KUKA KRL program: MyProgram_110().src

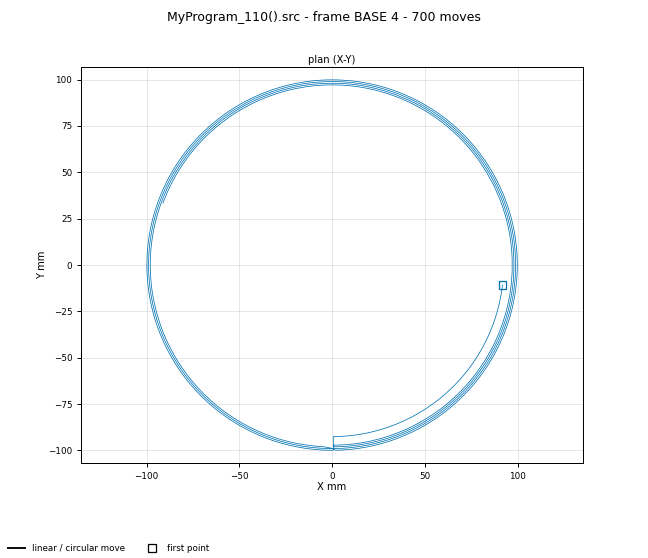
[picture p0: tool path of MyProgram_110().src in frame BASE 4, 700 of 700 moves have a stored position in this frame; points joined in program order, loops and branches not executed]
&ACCESS RVP
&REL 1
&PARAM TEMPLATE = C:\KRC\Roboter\Template\vorgabe
&PARAM EDITMASK = *
DEF MyProgram_110()
; ---- Setting reference (Base) ----
$BASE = BASE_DATA[4]

; --------------------------
; ---- Setting tool (TCP) ----
$TOOL = TOOL_DATA[3]
; --------------------------

$VEL.CP = VEL_APROX_PRINT
Startdeposition()
$VEL.CP = VEL_PRINT
LIN {X 91.8792,Y -10.8484,Z 96,A -11.884,B 24.923,C -2.0263,E1 25.1586,E2 97.0234} C_DIS
LIN {X 91.5181,Y -13.5726,Z 96,A -13.5745,B 24.9234,C -2.0212,E1 25.1579,E2 98.7159} C_DIS
LIN {X 91.0731,Y -16.2835,Z 96,A -15.3127,B 24.9239,C -2.0144,E1 25.1571,E2 100.46} C_DIS
LIN {X 90.5157,Y -19.1486,Z 96,A -17.2609,B 24.9247,C -2.0034,E1 25.156,E2 102.4228} C_DIS
LIN {X 89.7406,Y -22.5028,Z 96,A -19.3635,B 24.9252,C -1.9977,E1 25.1546,E2 104.5265} C_DIS
LIN {X 88.9858,Y -25.3177,Z 96,A -21.051,B 24.9252,C -1.9964,E1 25.1534,E2 106.2075} C_DIS
LIN {X 88.0495,Y -28.4034,Z 96,A -23.0482,B 24.9257,C -1.9901,E1 25.1517,E2 108.2082} C_DIS
LIN {X 87.1124,Y -31.1642,Z 96,A -24.7456,B 24.9259,C -1.9885,E1 25.1502,E2 109.8999} C_DIS
LIN {X 86.1483,Y -33.7335,Z 96,A -26.4825,B 24.9264,C -1.9819,E1 25.1484,E2 111.6427} C_DIS
LIN {X 85.0444,Y -36.4307,Z 96,A -28.2267,B 24.9266,C -1.9786,E1 25.1466,E2 113.3851} C_DIS
LIN {X 83.8742,Y -39.0457,Z 96,A -30.1195,B 24.9273,C -1.9689,E1 25.1444,E2 115.2905} C_DIS
LIN {X 82.3306,Y -42.2037,Z 96,A -32.231,B 24.9276,C -1.9648,E1 25.1417,E2 117.4003} C_DIS
LIN {X 80.8218,Y -45.0257,Z 96,A -34.1754,B 24.9279,C -1.9604,E1 25.1391,E2 119.345} C_DIS
LIN {X 79.3526,Y -47.5703,Z 96,A -35.9275,B 24.9282,C -1.9576,E1 25.1367,E2 121.0947} C_DIS
LIN {X 78.165,Y -49.4976,Z 96,A -37.5141,B 24.9289,C -1.9468,E1 25.1343,E2 122.6986} C_DIS
LIN {X 76.385,Y -52.2011,Z 96,A -39.5403,B 24.9294,C -1.9404,E1 25.1311,E2 124.7299} C_DIS
LIN {X 74.2916,Y -55.1408,Z 96,A -41.7416,B 24.9298,C -1.9355,E1 25.1275,E2 126.9321} C_DIS
LIN {X 72.2294,Y -57.816,Z 96,A -43.8281,B 24.9302,C -1.9302,E1 25.1239,E2 129.0215} C_DIS
LIN {X 70.1015,Y -60.3779,Z 96,A -45.7008,B 24.93,C -1.9317,E1 25.1205,E2 130.8819} C_DIS
LIN {X 68.086,Y -62.64,Z 96,A -47.6453,B 24.9306,C -1.9245,E1 25.1169,E2 132.8349} C_DIS
LIN {X 65.7943,Y -65.0428,Z 96,A -49.6815,B 24.9309,C -1.9202,E1 25.1129,E2 134.8726} C_DIS
LIN {X 63.3926,Y -67.3857,Z 96,A -51.8033,B 24.9314,C -1.9136,E1 25.1086,E2 137.0011} C_DIS
LIN {X 60.815,Y -69.7209,Z 96,A -53.9021,B 24.9316,C -1.9106,E1 25.1043,E2 139.0986} C_DIS
LIN {X 58.2335,Y -71.891,Z 96,A -55.9751,B 24.9319,C -1.9065,E1 25.0998,E2 141.1733} C_DIS
LIN {X 55.635,Y -73.9203,Z 96,A -57.9461,B 24.9319,C -1.9047,E1 25.0955,E2 143.1413} C_DIS
LIN {X 53.2621,Y -75.65,Z 96,A -59.9459,B 24.9327,C -1.8944,E1 25.0909,E2 145.1585} C_DIS
LIN {X 50.4399,Y -77.5601,Z 96,A -62.0149,B 24.9329,C -1.8918,E1 25.0861,E2 147.2269} C_DIS
LIN {X 47.9711,Y -79.109,Z 96,A -63.6084,B 24.9326,C -1.896,E1 25.0823,E2 148.8054} C_DIS
LIN {X 45.886,Y -80.3367,Z 96,A -65.1676,B 24.933,C -1.8911,E1 25.0785,E2 150.3715} C_DIS
LIN {X 43.0135,Y -81.9104,Z 96,A -67.2008,B 24.9332,C -1.8874,E1 25.0735,E2 152.4075} C_DIS
LIN {X 40.0034,Y -83.4218,Z 96,A -69.2752,B 24.9334,C -1.8844,E1 25.0683,E2 154.4835} C_DIS
LIN {X 37.0509,Y -84.7744,Z 96,A -71.2544,B 24.9336,C -1.8825,E1 25.0633,E2 156.4623} C_DIS
LIN {X 34.7139,Y -85.758,Z 96,A -72.8404,B 24.9338,C -1.8797,E1 25.0592,E2 158.0513} C_DIS
LIN {X 31.7652,Y -86.8932,Z 96,A -74.7688,B 24.9338,C -1.878,E1 25.0541,E2 159.9795} C_DIS
LIN {X 29.468,Y -87.6989,Z 96,A -76.2248,B 24.9338,C -1.878,E1 25.0503,E2 161.4329} C_DIS
LIN {X 26.8544,Y -88.536,Z 96,A -78.1126,B 24.9345,C -1.8693,E1 25.0452,E2 163.3376} C_DIS
LIN {X 24.0508,Y -89.3366,Z 96,A -79.8048,B 24.9344,C -1.8713,E1 25.0407,E2 165.0223} C_DIS
LIN {X 21.1355,Y -90.0714,Z 96,A -81.4386,B 24.9339,C -1.8775,E1 25.0363,E2 166.6391} C_DIS
LIN {X 18.575,Y -90.6335,Z 96,A -83.2717,B 24.9345,C -1.8687,E1 25.0312,E2 168.4906} C_DIS
LIN {X 15.4389,Y -91.2202,Z 96,A -85.2579,B 24.9347,C -1.8668,E1 25.0258,E2 170.4792} C_DIS
LIN {X 12.4455,Y -91.6781,Z 96,A -87.2375,B 24.935,C -1.8619,E1 25.0203,E2 172.4688} C_DIS
LIN {X 9.5456,Y -92.0236,Z 96,A -88.9335,B 24.9348,C -1.8647,E1 25.0156,E2 174.1568} C_DIS
LIN {X 6.3282,Y -92.3007,Z 96,A -90.8986,B 24.9348,C -1.8649,E1 25.0101,E2 176.1204} C_DIS
LIN {X 3.3948,Y -92.4567,Z 96,A -92.6665,B 24.9348,C -1.866,E1 25.0052,E2 177.8853} C_DIS
LIN {X 0.6474,Y -92.5151,Z 96,A -93.6353,B 24.933,C -1.8907,E1 25.0027,E2 178.7952} C_DIS
Enddeposition()
LIN {X 0.6893,Y -99.8812,Z 97,A -93.5468,B 24.9411,C -1.7731,E1 25.0021,E2 178.9855} C_DIS
Startdeposition()
$VEL.CP = VEL_PRINT
LIN {X -3.3316,Y -99.8302,Z 97,A -96.4114,B 24.9425,C -1.7518,E1 24.994,E2 181.9007} C_DIS
LIN {X -6.1252,Y -99.6993,Z 97,A -98.0149,B 24.9425,C -1.7518,E1 24.9895,E2 183.505} C_DIS
LIN {X -8.5701,Y -99.519,Z 97,A -99.4216,B 24.9425,C -1.7518,E1 24.9856,E2 184.9122} C_DIS
LIN {X -12.2273,Y -99.1361,Z 97,A -101.5316,B 24.9425,C -1.752,E1 24.9798,E2 187.0229} C_DIS
LIN {X -14.6565,Y -98.8061,Z 97,A -102.9384,B 24.9425,C -1.7523,E1 24.9759,E2 188.4302} C_DIS
LIN {X -17.0769,Y -98.4167,Z 97,A -104.3453,B 24.9425,C -1.7527,E1 24.972,E2 189.8375} C_DIS
LIN {X -19.1482,Y -98.0332,Z 97,A -105.7373,B 24.9428,C -1.7465,E1 24.9681,E2 191.2458} C_DIS
LIN {X -22.5412,Y -97.3087,Z 97,A -107.5895,B 24.9424,C -1.7524,E1 24.9631,E2 193.0862} C_DIS
LIN {X -25.1236,Y -96.6745,Z 97,A -109.0745,B 24.9423,C -1.7547,E1 24.9591,E2 194.5678} C_DIS
LIN {X -27.3483,Y -96.0686,Z 97,A -110.4263,B 24.9423,C -1.7545,E1 24.9554,E2 195.9222} C_DIS
LIN {X -29.8369,Y -95.3253,Z 97,A -111.931,B 24.9423,C -1.7551,E1 24.9514,E2 197.4282} C_DIS
LIN {X -32.4944,Y -94.4541,Z 97,A -113.4981,B 24.9421,C -1.7577,E1 24.9473,E2 198.9921} C_DIS
LIN {X -34.8026,Y -93.6282,Z 97,A -114.907,B 24.9421,C -1.7588,E1 24.9436,E2 200.4011} C_DIS
LIN {X -37.0899,Y -92.7459,Z 97,A -116.3162,B 24.9419,C -1.7601,E1 24.9399,E2 201.8103} C_DIS
LIN {X -39.3548,Y -91.8078,Z 97,A -117.7257,B 24.9419,C -1.7614,E1 24.9363,E2 203.2199} C_DIS
LIN {X -42.5339,Y -90.3777,Z 97,A -119.7156,B 24.9417,C -1.764,E1 24.9312,E2 205.2085} C_DIS
LIN {X -44.9105,Y -89.2217,Z 97,A -121.2502,B 24.9417,C -1.7652,E1 24.9274,E2 206.7443} C_DIS
LIN {X -46.7812,Y -88.2535,Z 97,A -122.502,B 24.9416,C -1.7652,E1 24.9243,E2 207.9994} C_DIS
LIN {X -49.8056,Y -86.5823,Z 97,A -124.4959,B 24.9414,C -1.7675,E1 24.9194,E2 209.9937} C_DIS
LIN {X -52.1049,Y -85.2188,Z 97,A -125.9883,B 24.9412,C -1.7712,E1 24.9159,E2 211.4819} C_DIS
LIN {X -54.1806,Y -83.9144,Z 97,A -127.3996,B 24.9411,C -1.7732,E1 24.9126,E2 212.893} C_DIS
LIN {X -56.5094,Y -82.366,Z 97,A -129.0091,B 24.9409,C -1.7756,E1 24.9088,E2 214.5022} C_DIS
LIN {X -59.2243,Y -80.4341,Z 97,A -130.8958,B 24.9406,C -1.7797,E1 24.9046,E2 216.3857} C_DIS
LIN {X -61.4538,Y -78.7458,Z 97,A -132.5381,B 24.9406,C -1.7812,E1 24.9009,E2 218.0304} C_DIS
LIN {X -64.3106,Y -76.4305,Z 97,A -134.6562,B 24.9403,C -1.7848,E1 24.8963,E2 220.1478} C_DIS
LIN {X -67.0802,Y -74.0116,Z 97,A -136.7744,B 24.94,C -1.7887,E1 24.8919,E2 222.2654} C_DIS
LIN {X -69.5104,Y -71.7319,Z 97,A -138.6946,B 24.9398,C -1.7923,E1 24.888,E2 224.1848} C_DIS
LIN {X -71.4924,Y -69.7589,Z 97,A -140.3062,B 24.9396,C -1.7954,E1 24.8849,E2 225.7958} C_DIS
LIN {X -73.1828,Y -67.9834,Z 97,A -141.7193,B 24.9394,C -1.7983,E1 24.8822,E2 227.2083} C_DIS
LIN {X -74.599,Y -66.424,Z 97,A -142.9737,B 24.9394,C -1.7994,E1 24.8798,E2 228.4656} C_DIS
LIN {X -76.4305,Y -64.3106,Z 97,A -144.6779,B 24.9393,C -1.7996,E1 24.8767,E2 230.177} C_DIS
LIN {X -78.3804,Y -61.9161,Z 97,A -146.3783,B 24.9388,C -1.8063,E1 24.8737,E2 231.8695} C_DIS
LIN {X -80.2302,Y -59.5028,Z 97,A -148.0798,B 24.9385,C -1.812,E1 24.8709,E2 233.5657} C_DIS
LIN {X -81.6663,Y -57.5159,Z 97,A -149.4938,B 24.9382,C -1.8152,E1 24.8686,E2 234.9788} C_DIS
LIN {X -83.728,Y -54.471,Z 97,A -151.615,B 24.9379,C -1.8202,E1 24.8653,E2 237.0988} C_DIS
LIN {X -85.0396,Y -52.3998,Z 97,A -153.1721,B 24.938,C -1.8187,E1 24.863,E2 238.6673} C_DIS
LIN {X -86.6472,Y -49.6927,Z 97,A -154.9304,B 24.9376,C -1.8252,E1 24.8605,E2 240.4193} C_DIS
LIN {X -87.9282,Y -47.3899,Z 97,A -156.4067,B 24.9372,C -1.8305,E1 24.8585,E2 241.8907} C_DIS
LIN {X -89.6129,Y -44.1214,Z 97,A -158.529,B 24.9368,C -1.8359,E1 24.8559,E2 244.0115} C_DIS
LIN {X -90.6687,Y -41.9089,Z 97,A -159.944,B 24.9366,C -1.8395,E1 24.8542,E2 245.4255} C_DIS
LIN {X -91.8078,Y -39.3548,Z 97,A -161.5178,B 24.9362,C -1.8451,E1 24.8524,E2 246.9947} C_DIS
LIN {X -92.7459,Y -37.0899,Z 97,A -162.9333,B 24.9359,C -1.8489,E1 24.8509,E2 248.4091} C_DIS
LIN {X -93.93,Y -33.9752,Z 97,A -164.8971,B 24.9357,C -1.8527,E1 24.849,E2 250.3747} C_DIS
LIN {X -94.7355,Y -31.6598,Z 97,A -166.4556,B 24.9357,C -1.8518,E1 24.8476,E2 251.9443} C_DIS
LIN {X -95.7659,Y -28.3899,Z 97,A -168.3053,B 24.935,C -1.8617,E1 24.8461,E2 253.7812} C_DIS
LIN {X -96.5386,Y -25.6432,Z 97,A -170.0582,B 24.935,C -1.8628,E1 24.8448,E2 255.5417} C_DIS
LIN {X -97.3463,Y -22.3787,Z 97,A -171.9204,B 24.9344,C -1.8709,E1 24.8436,E2 257.3953} C_DIS
LIN {X -98.1224,Y -18.6848,Z 97,A -174.0326,B 24.9338,C -1.8794,E1 24.8424,E2 259.4997} C_DIS
LIN {X -98.5387,Y -16.3472,Z 97,A -175.4664,B 24.9337,C -1.8813,E1 24.8418,E2 260.9376} C_DIS
LIN {X -98.93,Y -13.7846,Z 97,A -176.9308,B 24.9333,C -1.8867,E1 24.8412,E2 262.3978} C_DIS
LIN {X -99.2385,Y -11.3525,Z 97,A -178.3299,B 24.9329,C -1.8914,E1 24.8407,E2 263.7941} C_DIS
LIN {X -99.519,Y -8.5701,Z 97,A -179.922,B 24.9325,C -1.8969,E1 24.8403,E2 265.3826} C_DIS
LIN {X -99.7479,Y -5.2458,Z 97,A 178.1129,B 24.9322,C -1.9012,E1 24.84,E2 267.3492} C_DIS
LIN {X -99.8572,Y -2.4514,Z 97,A 176.5378,B 24.9318,C -1.9073,E1 24.8398,E2 268.9193} C_DIS
LIN {X -99.8873,Y -0.1345,Z 97,A 175.1594,B 24.9316,C -1.9099,E1 24.8398,E2 270.2997} C_DIS
LIN {X -99.8302,Y 3.3316,Z 97,A 173.1964,B 24.9311,C -1.9172,E1 24.8399,E2 272.2572} C_DIS
LIN {X -99.6993,Y 6.1252,Z 97,A 171.5813,B 24.9307,C -1.922,E1 24.8401,E2 273.8706} C_DIS
LIN {X -99.519,Y 8.5701,Z 97,A 170.1647,B 24.9304,C -1.9262,E1 24.8405,E2 275.2858} C_DIS
LIN {X -99.2385,Y 11.3525,Z 97,A 168.463,B 24.9304,C -1.9281,E1 24.841,E2 276.993} C_DIS
LIN {X -98.8061,Y 14.6565,Z 97,A 166.6246,B 24.9297,C -1.9367,E1 24.8417,E2 278.822} C_DIS
LIN {X -98.3065,Y 17.6896,Z 97,A 164.7927,B 24.9294,C -1.9401,E1 24.8425,E2 280.6566} C_DIS
LIN {X -97.7215,Y 20.6878,Z 97,A 162.8875,B 24.9294,C -1.9406,E1 24.8436,E2 282.5719} C_DIS
LIN {X -96.9756,Y 23.9354,Z 97,A 161.1593,B 24.9285,C -1.9527,E1 24.8447,E2 284.2812} C_DIS
LIN {X -96.269,Y 26.6412,Z 97,A 159.544,B 24.9282,C -1.9574,E1 24.8459,E2 285.8947} C_DIS
LIN {X -95.3253,Y 29.8369,Z 97,A 157.579,B 24.9279,C -1.9616,E1 24.8474,E2 287.861} C_DIS
LIN {X -94.5644,Y 32.1674,Z 97,A 156.1633,B 24.9276,C -1.9657,E1 24.8487,E2 289.2751} C_DIS
LIN {X -93.6282,Y 34.8026,Z 97,A 154.5885,B 24.9271,C -1.9716,E1 24.8502,E2 290.8447} C_DIS
LIN {X -92.4139,Y 37.9056,Z 97,A 152.6238,B 24.9268,C -1.9757,E1 24.8522,E2 292.8106} C_DIS
LIN {X -91.3179,Y 40.4784,Z 97,A 151.049,B 24.9264,C -1.9815,E1 24.854,E2 294.3802} C_DIS
LIN {X -90.297,Y 42.7073,Z 97,A 149.4906,B 24.9264,C -1.9806,E1 24.8558,E2 295.9492} C_DIS
LIN {X -88.9363,Y 45.469,Z 97,A 147.7517,B 24.926,C -1.9868,E1 24.858,E2 297.6827} C_DIS
LIN {X -87.5083,Y 48.164,Z 97,A 146.0951,B 24.9254,C -1.995,E1 24.8602,E2 299.3286} C_DIS
LIN {X -86.2999,Y 50.2971,Z 97,A 144.4843,B 24.9256,C -1.9922,E1 24.8624,E2 300.9544} C_DIS
LIN {X -84.573,Y 53.1468,Z 97,A 142.7567,B 24.9247,C -2.0038,E1 24.8649,E2 302.6632} C_DIS
LIN {X -83.2432,Y 55.2063,Z 97,A 141.3017,B 24.9245,C -2.0061,E1 24.8672,E2 304.12} C_DIS
LIN {X -81.8633,Y 57.2326,Z 97,A 139.8868,B 24.9243,C -2.0097,E1 24.8694,E2 305.5333} C_DIS
LIN {X -80.2302,Y 59.5028,Z 97,A 138.3134,B 24.9239,C -2.0151,E1 24.872,E2 307.1016} C_DIS
LIN {X -78.3291,Y 61.981,Z 97,A 136.4683,B 24.9236,C -2.0181,E1 24.8752,E2 308.9483} C_DIS
LIN {X -76.4305,Y 64.3106,Z 97,A 134.7774,B 24.9232,C -2.0236,E1 24.8782,E2 310.6338} C_DIS
LIN {X -74.8292,Y 66.1669,Z 97,A 133.3632,B 24.923,C -2.0269,E1 24.8808,E2 312.0463} C_DIS
LIN {X -72.6112,Y 68.5913,Z 97,A 131.4603,B 24.9226,C -2.0311,E1 24.8844,E2 313.9478} C_DIS
LIN {X -70.8735,Y 70.3855,Z 97,A 129.9872,B 24.9225,C -2.0332,E1 24.8872,E2 315.4222} C_DIS
LIN {X -68.8763,Y 72.3431,Z 97,A 128.4152,B 24.9221,C -2.0381,E1 24.8904,E2 316.9891} C_DIS
LIN {X -66.424,Y 74.599,Z 97,A 126.4537,B 24.9219,C -2.0408,E1 24.8944,E2 318.9521} C_DIS
LIN {X -64.3657,Y 76.3835,Z 97,A 124.9346,B 24.9215,C -2.0458,E1 24.8977,E2 320.4652} C_DIS
LIN {X -62.4573,Y 77.9518,Z 97,A 123.4987,B 24.9213,C -2.0482,E1 24.9008,E2 321.9007} C_DIS
LIN {X -60.7562,Y 79.2833,Z 97,A 122.2147,B 24.9213,C -2.0493,E1 24.9036,E2 323.1867} C_DIS
LIN {X -58.5138,Y 80.9544,Z 97,A 120.6435,B 24.9209,C -2.0537,E1 24.9071,E2 324.753} C_DIS
LIN {X -55.7801,Y 82.8598,Z 97,A 118.6836,B 24.9207,C -2.0559,E1 24.9116,E2 326.7143} C_DIS
LIN {X -53.7317,Y 84.2025,Z 97,A 117.2723,B 24.9206,C -2.0583,E1 24.9149,E2 328.1244} C_DIS
LIN {X -51.6472,Y 85.497,Z 97,A 115.8594,B 24.9204,C -2.0607,E1 24.9183,E2 329.5359} C_DIS
LIN {X -49.5335,Y 86.7387,Z 97,A 114.4477,B 24.9202,C -2.0631,E1 24.9217,E2 330.9463} C_DIS
LIN {X -46.3073,Y 88.5031,Z 97,A 112.3707,B 24.9198,C -2.0677,E1 24.9268,E2 333.018} C_DIS
LIN {X -44.2378,Y 89.5552,Z 97,A 110.9639,B 24.9198,C -2.0673,E1 24.9303,E2 334.4296} C_DIS
LIN {X -41.9089,Y 90.6687,Z 97,A 109.5082,B 24.9196,C -2.0704,E1 24.934,E2 335.8815} C_DIS
LIN {X -38.5432,Y 92.1498,Z 97,A 107.3922,B 24.9194,C -2.0733,E1 24.9394,E2 337.9958} C_DIS
LIN {X -35.1253,Y 93.506,Z 97,A 105.3167,B 24.9191,C -2.0773,E1 24.9448,E2 340.0661} C_DIS
LIN {X -32.9512,Y 94.2938,Z 97,A 103.9603,B 24.9191,C -2.0779,E1 24.9484,E2 341.4237} C_DIS
LIN {X -30.4949,Y 95.1169,Z 97,A 102.4565,B 24.9189,C -2.0791,E1 24.9524,E2 342.9275} C_DIS
LIN {X -27.8206,Y 95.9348,Z 97,A 100.8884,B 24.9187,C -2.0821,E1 24.9566,E2 344.4912} C_DIS
LIN {X -25.4578,Y 96.5886,Z 97,A 99.4792,B 24.9186,C -2.0834,E1 24.9604,E2 345.8993} C_DIS
LIN {X -23.0798,Y 97.1843,Z 97,A 98.0702,B 24.9186,C -2.0847,E1 24.9642,E2 347.3073} C_DIS
LIN {X -20.6878,Y 97.7215,Z 97,A 96.6609,B 24.9184,C -2.0858,E1 24.968,E2 348.7157} C_DIS
LIN {X -18.2834,Y 98.1997,Z 97,A 95.2523,B 24.9184,C -2.0868,E1 24.9719,E2 350.1233} C_DIS
LIN {X -14.9975,Y 98.7534,Z 97,A 93.3379,B 24.9182,C -2.0881,E1 24.9771,E2 352.0365} C_DIS
LIN {X -12.2273,Y 99.1361,Z 97,A 91.7317,B 24.9182,C -2.089,E1 24.9816,E2 353.6418} C_DIS
LIN {X -9.7907,Y 99.4063,Z 97,A 90.324,B 24.9182,C -2.0897,E1 24.9855,E2 355.0487} C_DIS
LIN {X -6.4695,Y 99.676,Z 97,A 88.4105,B 24.918,C -2.0905,E1 24.9908,E2 356.9611} C_DIS
LIN {X -3.6766,Y 99.8196,Z 97,A 86.8052,B 24.918,C -2.0909,E1 24.9953,E2 358.5656} C_DIS
LIN {X -1.2258,Y 99.8798,Z 97,A 85.2558,B 24.9184,C -2.0861,E1 24.9997,E2 360.1266} C_DIS
LIN {X 1.9588,Y 99.8663,Z 97,A 83.5428,B 24.918,C -2.0906,E1 25.0044,E2 361.8289} C_DIS
LIN {X 4.5565,Y 99.7818,Z 97,A 82.0396,B 24.918,C -2.0902,E1 25.0086,E2 363.3325} C_DIS
LIN {X 7.3482,Y 99.6166,Z 97,A 80.4755,B 24.918,C -2.0916,E1 25.013,E2 364.8926} C_DIS
LIN {X 9.447,Y 99.438,Z 97,A 79.2675,B 24.918,C -2.0916,E1 25.0163,E2 366.1001} C_DIS
LIN {X 12.2273,Y 99.1361,Z 97,A 77.6636,B 24.918,C -2.0912,E1 25.0208,E2 367.7035} C_DIS
LIN {X 14.6565,Y 98.8061,Z 97,A 76.2582,B 24.918,C -2.0909,E1 25.0246,E2 369.1085} C_DIS
LIN {X 17.67,Y 98.31,Z 97,A 74.4468,B 24.9182,C -2.0881,E1 25.0296,E2 370.9245} C_DIS
LIN {X 20.3497,Y 97.7908,Z 97,A 72.9037,B 24.9182,C -2.0883,E1 25.0339,E2 372.4654} C_DIS
LIN {X 22.7435,Y 97.262,Z 97,A 71.4988,B 24.9182,C -2.0876,E1 25.0377,E2 373.87} C_DIS
LIN {X 26.3081,Y 96.359,Z 97,A 69.4324,B 24.9182,C -2.0879,E1 25.0433,E2 375.9326} C_DIS
LIN {X 28.9957,Y 95.5862,Z 97,A 67.8306,B 24.9183,C -2.0868,E1 25.0476,E2 377.5342} C_DIS
LIN {X 31.6598,Y 94.7355,Z 97,A 66.1296,B 24.9187,C -2.0819,E1 25.0521,E2 379.2436} C_DIS
LIN {X 34.4784,Y 93.7465,Z 97,A 64.5392,B 24.9185,C -2.0849,E1 25.0562,E2 380.8235} C_DIS
LIN {X 37.0899,Y 92.7459,Z 97,A 62.9184,B 24.9187,C -2.0827,E1 25.0605,E2 382.446} C_DIS
LIN {X 39.3548,Y 91.8078,Z 97,A 61.5154,B 24.9187,C -2.0813,E1 25.0641,E2 383.8489} C_DIS
LIN {X 42.7073,Y 90.297,Z 97,A 59.4115,B 24.9189,C -2.0791,E1 25.0694,E2 385.9529} C_DIS
LIN {X 44.9105,Y 89.2217,Z 97,A 58.0088,B 24.9191,C -2.0775,E1 25.0729,E2 387.3556} C_DIS
LIN {X 47.0865,Y 88.0927,Z 97,A 56.6068,B 24.9191,C -2.0758,E1 25.0764,E2 388.7577} C_DIS
LIN {X 49.5335,Y 86.7387,Z 97,A 54.9133,B 24.9196,C -2.0702,E1 25.0805,E2 390.4595} C_DIS
LIN {X 52.3998,Y 85.0396,Z 97,A 53.1022,B 24.9196,C -2.0711,E1 25.0848,E2 392.2627} C_DIS
LIN {X 55.2063,Y 83.2432,Z 97,A 51.1576,B 24.9199,C -2.0668,E1 25.0894,E2 394.2111} C_DIS
LIN {X 57.5159,Y 81.6663,Z 97,A 49.3901,B 24.9206,C -2.0579,E1 25.0935,E2 395.9937} C_DIS
LIN {X 60.2069,Y 79.7012,Z 97,A 47.6949,B 24.9202,C -2.0628,E1 25.0973,E2 397.6711} C_DIS
LIN {X 62.1448,Y 78.1997,Z 97,A 46.2543,B 24.9205,C -2.0589,E1 25.1004,E2 399.1156} C_DIS
LIN {X 64.7268,Y 76.0758,Z 97,A 44.3079,B 24.9209,C -2.0542,E1 25.1046,E2 401.0657} C_DIS
LIN {X 66.8231,Y 74.2418,Z 97,A 42.7537,B 24.9209,C -2.0527,E1 25.1079,E2 402.6173} C_DIS
LIN {X 68.6249,Y 72.5795,Z 97,A 41.3536,B 24.9212,C -2.05,E1 25.1107,E2 404.0179} C_DIS
LIN {X 70.3855,Y 70.8735,Z 97,A 39.9537,B 24.9214,C -2.0473,E1 25.1135,E2 405.4184} C_DIS
LIN {X 72.3431,Y 68.8763,Z 97,A 38.3968,B 24.9215,C -2.0456,E1 25.1165,E2 406.9726} C_DIS
LIN {X 74.0116,Y 67.0802,Z 97,A 36.9977,B 24.9218,C -2.0428,E1 25.1192,E2 408.3723} C_DIS
LIN {X 75.9593,Y 64.8636,Z 97,A 35.2228,B 24.9223,C -2.0357,E1 25.1224,E2 410.1559} C_DIS
LIN {X 77.9857,Y 62.4155,Z 97,A 33.4998,B 24.9223,C -2.0353,E1 25.1255,E2 411.8718} C_DIS
LIN {X 79.7012,Y 60.2069,Z 97,A 31.8106,B 24.9229,C -2.0281,E1 25.1283,E2 413.5701} C_DIS
LIN {X 81.4659,Y 57.7968,Z 97,A 30.16,B 24.923,C -2.0263,E1 25.131,E2 415.2169} C_DIS
LIN {X 82.8598,Y 55.7801,Z 97,A 28.7616,B 24.9233,C -2.023,E1 25.1332,E2 416.6162} C_DIS
LIN {X 84.3901,Y 53.4395,Z 97,A 27.2062,B 24.9234,C -2.0207,E1 25.1356,E2 418.1691} C_DIS
LIN {X 86.2999,Y 50.2971,Z 97,A 25.1088,B 24.9238,C -2.0156,E1 25.1386,E2 420.2679} C_DIS
LIN {X 87.5083,Y 48.164,Z 97,A 23.711,B 24.9241,C -2.0121,E1 25.1405,E2 421.6667} C_DIS
LIN {X 89.0647,Y 45.2177,Z 97,A 21.7712,B 24.9246,C -2.0057,E1 25.143,E2 423.6113} C_DIS
LIN {X 90.5278,Y 42.2116,Z 97,A 19.8287,B 24.925,C -1.9994,E1 25.1454,E2 425.5583} C_DIS
LIN {X 91.6699,Y 39.6711,Z 97,A 18.317,B 24.9251,C -1.9982,E1 25.1471,E2 427.0645} C_DIS
LIN {X 92.7341,Y 37.1188,Z 97,A 16.7403,B 24.9255,C -1.9939,E1 25.1487,E2 428.6426} C_DIS
LIN {X 93.6282,Y 34.8026,Z 97,A 15.3257,B 24.9257,C -1.9901,E1 25.1501,E2 430.0583} C_DIS
LIN {X 94.7355,Y 31.6598,Z 97,A 13.3868,B 24.9262,C -1.9834,E1 25.1519,E2 432.0022} C_DIS
LIN {X 95.8366,Y 28.1514,Z 97,A 11.3309,B 24.9266,C -1.9791,E1 25.1536,E2 434.0564} C_DIS
LIN {X 96.439,Y 26.0118,Z 97,A 9.9684,B 24.9271,C -1.9718,E1 25.1546,E2 435.4285} C_DIS
LIN {X 97.1843,Y 23.0798,Z 97,A 8.1279,B 24.9278,C -1.9622,E1 25.1558,E2 437.2809} C_DIS
LIN {X 97.8986,Y 19.8251,Z 97,A 6.4419,B 24.9276,C -1.9653,E1 25.1568,E2 438.9498} C_DIS
LIN {X 98.3556,Y 17.4166,Z 97,A 5.0056,B 24.928,C -1.9597,E1 25.1575,E2 440.3909} C_DIS
LIN {X 98.93,Y 13.7846,Z 97,A 2.9105,B 24.9284,C -1.9536,E1 25.1584,E2 442.488} C_DIS
LIN {X 99.3146,Y 10.6666,Z 97,A 1.0621,B 24.929,C -1.946,E1 25.159,E2 444.3434} C_DIS
LIN {X 99.5891,Y 7.6922,Z 97,A -0.5411,B 24.929,C -1.945,E1 25.1594,E2 445.9396} C_DIS
LIN {X 99.7479,Y 5.2458,Z 97,A -1.9333,B 24.9294,C -1.941,E1 25.1596,E2 447.3328} C_DIS
LIN {X 99.8572,Y 2.4514,Z 97,A -3.5306,B 24.9297,C -1.9361,E1 25.1598,E2 448.9321} C_DIS
LIN {X 99.8873,Y 0.1345,Z 97,A -4.8678,B 24.9301,C -1.9315,E1 25.1598,E2 450.2722} C_DIS
LIN {X 99.8635,Y -2.1063,Z 97,A -6.1269,B 24.9303,C -1.9285,E1 25.1598,E2 451.5311} C_DIS
LIN {X 99.7818,Y -4.5565,Z 97,A -7.563,B 24.9307,C -1.9227,E1 25.1596,E2 452.9722} C_DIS
LIN {X 99.6166,Y -7.3482,Z 97,A -9.1164,B 24.9309,C -1.9196,E1 25.1593,E2 454.5238} C_DIS
LIN {X 99.438,Y -9.447,Z 97,A -10.4969,B 24.9317,C -1.9088,E1 25.1589,E2 455.9215} C_DIS
LIN {X 99.0553,Y -12.8503,Z 97,A -12.3697,B 24.9319,C -1.9061,E1 25.1583,E2 457.7895} C_DIS
LIN {X 98.5619,Y -16.2083,Z 97,A -14.301,B 24.9323,C -1.9005,E1 25.1575,E2 459.7228} C_DIS
LIN {X 98.0332,Y -19.1482,Z 97,A -15.9415,B 24.9325,C -1.8979,E1 25.1566,E2 461.3598} C_DIS
LIN {X 97.5338,Y -21.5483,Z 97,A -17.3382,B 24.9328,C -1.8938,E1 25.1558,E2 462.7581} C_DIS
LIN {X 96.9756,Y -23.9354,Z 97,A -18.7347,B 24.9331,C -1.8897,E1 25.1549,E2 464.1561} C_DIS
LIN {X 96.1242,Y -27.1522,Z 97,A -20.6715,B 24.9336,C -1.8825,E1 25.1535,E2 466.0987} C_DIS
LIN {X 95.3253,Y -29.8369,Z 97,A -22.2263,B 24.9338,C -1.8796,E1 25.1522,E2 467.6517} C_DIS
LIN {X 94.534,Y -32.2576,Z 97,A -23.6266,B 24.9339,C -1.8774,E1 25.151,E2 469.0491} C_DIS
LIN {X 93.6282,Y -34.8026,Z 97,A -25.1768,B 24.9343,C -1.8726,E1 25.1495,E2 470.6021} C_DIS
LIN {X 92.8322,Y -36.8703,Z 97,A -26.4272,B 24.9345,C -1.8695,E1 25.1482,E2 471.8528} C_DIS
LIN {X 91.8078,Y -39.3548,Z 97,A -27.9706,B 24.9348,C -1.8647,E1 25.1465,E2 473.3991} C_DIS
LIN {X 90.297,Y -42.7073,Z 97,A -30.2071,B 24.9356,C -1.8532,E1 25.1439,E2 475.6505} C_DIS
LIN {X 88.8915,Y -45.5567,Z 97,A -31.9062,B 24.9356,C -1.8528,E1 25.1418,E2 477.3417} C_DIS
LIN {X 87.5083,Y -48.164,Z 97,A -33.5594,B 24.9359,C -1.8493,E1 25.1396,E2 478.9942} C_DIS
LIN {X 86.2999,Y -50.2971,Z 97,A -34.9566,B 24.9361,C -1.8456,E1 25.1377,E2 480.393} C_DIS
LIN {X 84.573,Y -53.1468,Z 97,A -36.8561,B 24.9365,C -1.8406,E1 25.1349,E2 482.2946} C_DIS
LIN {X 83.2432,Y -55.2063,Z 97,A -38.2934,B 24.9369,C -1.8354,E1 25.1327,E2 483.737} C_DIS
LIN {X 81.6663,Y -57.5159,Z 97,A -39.8484,B 24.937,C -1.8329,E1 25.1302,E2 485.2903} C_DIS
LIN {X 79.7093,Y -60.1963,Z 97,A -41.7834,B 24.9375,C -1.8265,E1 25.127,E2 487.2311} C_DIS
LIN {X 78.1997,Y -62.1448,Z 97,A -43.3276,B 24.9381,C -1.8176,E1 25.1243,E2 488.7892} C_DIS
LIN {X 75.9775,Y -64.8423,Z 97,A -45.1758,B 24.9381,C -1.8185,E1 25.121,E2 490.6266} C_DIS
LIN {X 74.0116,Y -67.0802,Z 97,A -46.8391,B 24.9381,C -1.8159,E1 25.1179,E2 492.2887} C_DIS
LIN {X 71.7319,Y -69.5104,Z 97,A -48.7404,B 24.9385,C -1.8116,E1 25.1143,E2 494.1919} C_DIS
LIN {X 69.7589,Y -71.4924,Z 97,A -50.3359,B 24.9387,C -1.808,E1 25.1111,E2 495.7892} C_DIS
LIN {X 68.1601,Y -73.0167,Z 97,A -51.6176,B 24.939,C -1.8044,E1 25.1085,E2 497.074} C_DIS
LIN {X 66.1669,Y -74.8292,Z 97,A -53.3189,B 24.9396,C -1.7947,E1 25.1049,E2 498.7915} C_DIS
LIN {X 63.6332,Y -76.9933,Z 97,A -55.0761,B 24.9396,C -1.7965,E1 25.1012,E2 500.5378} C_DIS
LIN {X 61.4538,Y -78.7458,Z 97,A -56.6329,B 24.9396,C -1.7948,E1 25.0978,E2 502.0927} C_DIS
LIN {X 59.5028,Y -80.2302,Z 97,A -58.0326,B 24.9398,C -1.7921,E1 25.0947,E2 503.4938} C_DIS
LIN {X 57.5159,Y -81.6663,Z 97,A -59.4327,B 24.94,C -1.7894,E1 25.0915,E2 504.8953} C_DIS
LIN {X 54.9039,Y -83.4425,Z 97,A -61.3177,B 24.9404,C -1.783,E1 25.0871,E2 506.7892} C_DIS
LIN {X 52.3998,Y -85.0396,Z 97,A -62.9335,B 24.9404,C -1.7831,E1 25.0833,E2 508.3995} C_DIS
LIN {X 50.2971,Y -86.2999,Z 97,A -64.3342,B 24.9406,C -1.7808,E1 25.0799,E2 509.8015} C_DIS
LIN {X 48.164,Y -87.5083,Z 97,A -65.735,B 24.9407,C -1.7785,E1 25.0765,E2 511.2035} C_DIS
LIN {X 46.002,Y -88.6639,Z 97,A -67.1357,B 24.9409,C -1.7763,E1 25.073,E2 512.6055} C_DIS
LIN {X 43.198,Y -90.0613,Z 97,A -68.9667,B 24.9411,C -1.7721,E1 25.0684,E2 514.4415} C_DIS
LIN {X 40.4784,Y -91.3179,Z 97,A -70.6392,B 24.9412,C -1.7712,E1 25.0642,E2 516.112} C_DIS
LIN {X 38.5432,Y -92.1498,Z 97,A -71.8837,B 24.9414,C -1.768,E1 25.061,E2 517.361} C_DIS
LIN {X 35.1253,Y -93.506,Z 97,A -73.9867,B 24.9416,C -1.7653,E1 25.0555,E2 519.4657} C_DIS
LIN {X 31.9939,Y -94.6229,Z 97,A -75.9307,B 24.9418,C -1.7615,E1 25.0503,E2 521.4149} C_DIS
LIN {X 29.5127,Y -95.4259,Z 97,A -77.4278,B 24.942,C -1.7597,E1 25.0464,E2 522.9136} C_DIS
LIN {X 25.8461,Y -96.4838,Z 97,A -79.5769,B 24.942,C -1.7588,E1 25.0406,E2 525.0612} C_DIS
LIN {X 23.0798,Y -97.1843,Z 97,A -81.1578,B 24.942,C -1.7593,E1 25.0363,E2 526.6387} C_DIS
LIN {X 20.6878,Y -97.7215,Z 97,A -82.5617,B 24.942,C -1.7581,E1 25.0325,E2 528.0435} C_DIS
LIN {X 18.2834,Y -98.1997,Z 97,A -83.9652,B 24.9421,C -1.757,E1 25.0286,E2 529.448} C_DIS
LIN {X 14.6565,Y -98.8061,Z 97,A -86.2735,B 24.9427,C -1.7479,E1 25.0222,E2 531.7754} C_DIS
LIN {X 11.3525,Y -99.2385,Z 97,A -88.0199,B 24.9424,C -1.753,E1 25.0174,E2 533.5086} C_DIS
LIN {X 8.5701,Y -99.519,Z 97,A -89.5823,B 24.9424,C -1.7537,E1 25.0131,E2 535.0684} C_DIS
LIN {X 5.2458,Y -99.7479,Z 97,A -91.5318,B 24.9425,C -1.7514,E1 25.0076,E2 537.0224} C_DIS
LIN {X 1.884,Y -99.8676,Z 97,A -93.4908,B 24.9426,C -1.7497,E1 25.0021,E2 538.985} C_DIS
LIN {X 1.884,Y -99.8676,Z 97,A -93.4908,B 24.9426,C -1.7497,E1 25.0021,E2 538.985} C_DIS
Enddeposition()
LIN {X 0.6835,Y -98.9739,Z 97,A -93.8467,B 24.9408,C -1.7778,E1 25.0013,E2 539.2743} C_DIS
Startdeposition()
$VEL.CP = VEL_PRINT
LIN {X 5.664,Y -98.8189,Z 97,A -90.6416,B 24.9399,C -1.7906,E1 25.0104,E2 536.0396} C_DIS
LIN {X 8.0719,Y -98.6514,Z 97,A -88.5771,B 24.9382,C -1.8165,E1 25.0163,E2 533.9149} C_DIS
LIN {X 11.6674,Y -98.291,Z 97,A -87.2398,B 24.94,C -1.7892,E1 25.0198,E2 532.6432} C_DIS
LIN {X 14.7111,Y -97.8825,Z 97,A -85.1348,B 24.9391,C -1.8027,E1 25.0257,E2 530.508} C_DIS
LIN {X 18.4972,Y -97.2375,Z 97,A -83.0849,B 24.9394,C -1.7979,E1 25.0313,E2 528.4717} C_DIS
LIN {X 21.4431,Y -96.631,Z 97,A -80.9548,B 24.9383,C -1.8144,E1 25.0372,E2 526.3055} C_DIS
LIN {X 25.1502,Y -95.7338,Z 97,A -78.9936,B 24.9388,C -1.8071,E1 25.0425,E2 524.3644} C_DIS
LIN {X 28.555,Y -94.7735,Z 97,A -77.0094,B 24.9388,C -1.8071,E1 25.0478,E2 522.3838} C_DIS
LIN {X 31.7611,Y -93.7469,Z 97,A -74.5566,B 24.9373,C -1.8289,E1 25.0544,E2 519.8839} C_DIS
LIN {X 35.2025,Y -92.5096,Z 97,A -73.0806,B 24.9388,C -1.807,E1 25.0581,E2 518.463} C_DIS
LIN {X 37.9038,Y -91.4378,Z 97,A -70.8744,B 24.9373,C -1.8296,E1 25.0639,E2 516.2082} C_DIS
LIN {X 42.0811,Y -89.5908,Z 97,A -68.749,B 24.9383,C -1.8136,E1 25.0692,E2 514.1262} C_DIS
LIN {X 46.1052,Y -87.5873,Z 97,A -66.0721,B 24.9379,C -1.8208,E1 25.0759,E2 511.4396} C_DIS
LIN {X 49.1629,Y -85.9084,Z 97,A -64.0723,B 24.9377,C -1.8236,E1 25.0808,E2 509.439} C_DIS
LIN {X 51.9174,Y -84.2743,Z 97,A -62.0938,B 24.9371,C -1.8319,E1 25.0855,E2 507.447} C_DIS
LIN {X 55.1663,Y -82.1831,Z 97,A -60.214,B 24.9377,C -1.8224,E1 25.0899,E2 505.596} C_DIS
LIN {X 57.0077,Y -80.9177,Z 97,A -58.6351,B 24.9368,C -1.8362,E1 25.0935,E2 503.9899} C_DIS
LIN {X 59.858,Y -78.8321,Z 97,A -56.7352,B 24.9368,C -1.8348,E1 25.0978,E2 502.1001} C_DIS
LIN {X 62.2733,Y -76.9368,Z 97,A -54.9996,B 24.9368,C -1.8371,E1 25.1016,E2 500.3655} C_DIS
LIN {X 64.6236,Y -74.9755,Z 97,A -53.2532,B 24.9365,C -1.84,E1 25.1053,E2 498.6189} C_DIS
LIN {X 67.0728,Y -72.7908,Z 97,A -51.1428,B 24.9356,C -1.8528,E1 25.1097,E2 496.4868} C_DIS
LIN {X 69.7831,Y -70.1971,Z 97,A -49.188,B 24.9359,C -1.8495,E1 25.1136,E2 494.5481} C_DIS
LIN {X 71.5892,Y -68.3552,Z 97,A -47.5463,B 24.9352,C -1.859,E1 25.1168,E2 492.8909} C_DIS
LIN {X 73.5521,Y -66.2375,Z 97,A -45.9105,B 24.935,C -1.8619,E1 25.1199,E2 491.2557} C_DIS
LIN {X 75.5108,Y -63.9953,Z 97,A -44.2428,B 24.9349,C -1.8641,E1 25.1229,E2 489.5903} C_DIS
LIN {X 77.5328,Y -61.5299,Z 97,A -42.3412,B 24.9344,C -1.8712,E1 25.1262,E2 487.6806} C_DIS
LIN {X 79.9171,Y -58.3994,Z 97,A -39.8903,B 24.9334,C -1.8844,E1 25.1304,E2 485.2105} C_DIS
LIN {X 82.5016,Y -54.688,Z 97,A -37.5417,B 24.9337,C -1.8809,E1 25.134,E2 482.8817} C_DIS
LIN {X 84.2377,Y -51.9762,Z 97,A -35.5305,B 24.9329,C -1.8921,E1 25.137,E2 480.8544} C_DIS
LIN {X 86.0633,Y -48.8935,Z 97,A -33.6836,B 24.9331,C -1.889,E1 25.1396,E2 479.0242} C_DIS
LIN {X 88.0812,Y -45.1547,Z 97,A -31.36,B 24.933,C -1.8908,E1 25.1426,E2 476.7086} C_DIS
LIN {X 89.5123,Y -42.2498,Z 97,A -28.2605,B 24.929,C -1.946,E1 25.1465,E2 473.4956} C_DIS
LIN {X 91.7324,Y -37.1807,Z 97,A -25.7407,B 24.9303,C -1.9279,E1 25.1491,E2 471.0322} C_DIS
LIN {X 93.1314,Y -33.5252,Z 97,A -23.9794,B 24.9313,C -1.9146,E1 25.1507,E2 469.3123} C_DIS
LIN {X 94.136,Y -30.5885,Z 97,A -22.0731,B 24.9306,C -1.9246,E1 25.1524,E2 467.393} C_DIS
LIN {X 95.3107,Y -26.7055,Z 97,A -19.8567,B 24.9304,C -1.9267,E1 25.1542,E2 465.1844} C_DIS
LIN {X 96.0937,Y -23.734,Z 97,A -17.9485,B 24.9296,C -1.9376,E1 25.1555,E2 463.2616} C_DIS
LIN {X 96.9548,Y -19.9246,Z 97,A -15.6346,B 24.9289,C -1.9469,E1 25.1569,E2 460.9391} C_DIS
LIN {X 97.5414,Y -16.8274,Z 97,A -13.7859,B 24.9284,C -1.9537,E1 25.1578,E2 459.0851} C_DIS
LIN {X 98.0665,Y -13.4321,Z 97,A -11.9219,B 24.9284,C -1.9551,E1 25.1585,E2 457.2289} C_DIS
LIN {X 98.7085,Y -7.3571,Z 97,A -8.5571,B 24.928,C -1.9596,E1 25.1594,E2 453.8735} C_DIS
LIN {X 98.8679,Y -4.755,Z 97,A -6.9038,B 24.9272,C -1.9702,E1 25.1597,E2 452.2048} C_DIS
LIN {X 98.9695,Y -1.5302,Z 97,A -4.2952,B 24.9245,C -2.0063,E1 25.1597,E2 449.5266} C_DIS
LIN {X 98.9327,Y 3.0897,Z 97,A -2.7289,B 24.9272,C -1.9701,E1 25.1597,E2 448.0551} C_DIS
LIN {X 98.607,Y 8.6093,Z 97,A 0.5739,B 24.9262,C -1.9843,E1 25.1591,E2 444.7383} C_DIS
LIN {X 98.2187,Y 12.2684,Z 97,A 2.8738,B 24.9252,C -1.9979,E1 25.1584,E2 442.4199} C_DIS
LIN {X 97.7818,Y 15.3623,Z 97,A 4.6515,B 24.9248,C -2.0024,E1 25.1576,E2 440.6422} C_DIS
LIN {X 97.1894,Y 18.7466,Z 97,A 6.6118,B 24.9244,C -2.0075,E1 25.1567,E2 438.6813} C_DIS
LIN {X 96.4599,Y 22.1974,Z 97,A 8.722,B 24.9238,C -2.0166,E1 25.1554,E2 436.5621} C_DIS
LIN {X 95.5557,Y 25.8133,Z 97,A 10.8015,B 24.9235,C -2.02,E1 25.1539,E2 434.4863} C_DIS
LIN {X 94.5448,Y 29.3003,Z 97,A 13.0513,B 24.9226,C -2.0323,E1 25.1521,E2 432.2203} C_DIS
LIN {X 93.5945,Y 32.2112,Z 97,A 14.7293,B 24.9224,C -2.0338,E1 25.1506,E2 430.5483} C_DIS
LIN {X 92.3789,Y 35.5478,Z 97,A 16.6614,B 24.9224,C -2.0349,E1 25.1487,E2 428.6244} C_DIS
LIN {X 91.2017,Y 38.4639,Z 97,A 18.4656,B 24.922,C -2.0396,E1 25.1468,E2 426.8192} C_DIS
LIN {X 89.3785,Y 42.5305,Z 97,A 21.1167,B 24.9212,C -2.0497,E1 25.1437,E2 424.1585} C_DIS
LIN {X 87.9585,Y 45.3947,Z 97,A 23.147,B 24.9203,C -2.062,E1 25.1411,E2 422.1099} C_DIS
LIN {X 85.7526,Y 49.434,Z 97,A 25.4968,B 24.9207,C -2.0567,E1 25.1379,E2 419.7848} C_DIS
LIN {X 84.0063,Y 52.3467,Z 97,A 27.4958,B 24.9202,C -2.0632,E1 25.135,E2 417.7806} C_DIS
LIN {X 82.0003,Y 55.4362,Z 97,A 29.5848,B 24.9199,C -2.067,E1 25.1318,E2 415.6931} C_DIS
LIN {X 80.3445,Y 57.8112,Z 97,A 31.1905,B 24.9198,C -2.0684,E1 25.1292,E2 414.0919} C_DIS
LIN {X 78.7593,Y 59.9544,Z 97,A 33.1122,B 24.9183,C -2.0871,E1 25.1259,E2 412.1352} C_DIS
LIN {X 75.5104,Y 63.9958,Z 97,A 35.7216,B 24.919,C -2.0788,E1 25.1214,E2 409.5575} C_DIS
LIN {X 73.3454,Y 66.4681,Z 97,A 37.7905,B 24.9181,C -2.0896,E1 25.1175,E2 407.4724} C_DIS
LIN {X 71.2811,Y 68.6748,Z 97,A 39.4405,B 24.9181,C -2.0896,E1 25.1143,E2 405.8295} C_DIS
LIN {X 69.1819,Y 70.7911,Z 97,A 41.5671,B 24.9166,C -2.1088,E1 25.11,E2 403.6663} C_DIS
LIN {X 64.7496,Y 74.8661,Z 97,A 44.6347,B 24.9173,C -2.0995,E1 25.1037,E2 400.633} C_DIS
LIN {X 62.8826,Y 76.4411,Z 97,A 46.1293,B 24.9169,C -2.1053,E1 25.1005,E2 399.1304} C_DIS
LIN {X 59.9441,Y 78.7673,Z 97,A 48.2124,B 24.9169,C -2.1059,E1 25.0959,E2 397.0535} C_DIS
LIN {X 57.5112,Y 80.5585,Z 97,A 49.6467,B 24.9175,C -2.0969,E1 25.0927,E2 395.6456} C_DIS
LIN {X 54.6922,Y 82.4988,Z 97,A 51.9013,B 24.9165,C -2.1106,E1 25.0875,E2 393.3662} C_DIS
LIN {X 51.8596,Y 84.3095,Z 97,A 53.983,B 24.9158,C -2.1188,E1 25.0825,E2 391.2719} C_DIS
LIN {X 48.4814,Y 86.2951,Z 97,A 56.0712,B 24.9161,C -2.1152,E1 25.0775,E2 389.1984} C_DIS
LIN {X 45.511,Y 87.8991,Z 97,A 57.9225,B 24.9161,C -2.1139,E1 25.0729,E2 387.3555} C_DIS
LIN {X 43.3891,Y 88.966,Z 97,A 59.4345,B 24.9156,C -2.1208,E1 25.0691,E2 385.8313} C_DIS
LIN {X 39.1996,Y 90.8887,Z 97,A 61.8773,B 24.9161,C -2.1153,E1 25.063,E2 383.4074} C_DIS
LIN {X 35.2288,Y 92.4997,Z 97,A 64.6046,B 24.9151,C -2.1271,E1 25.0558,E2 380.6584} C_DIS
LIN {X 31.4579,Y 93.8491,Z 97,A 66.6616,B 24.9158,C -2.1194,E1 25.0505,E2 378.6238} C_DIS
LIN {X 29.0692,Y 94.6164,Z 97,A 68.2479,B 24.9153,C -2.1255,E1 25.0462,E2 377.026} C_DIS
LIN {X 25.9595,Y 95.5162,Z 97,A 70.2584,B 24.9148,C -2.1318,E1 25.0408,E2 375.0037} C_DIS
LIN {X 22.8607,Y 96.3065,Z 97,A 72.2005,B 24.9144,C -2.1363,E1 25.0355,E2 373.054} C_DIS
LIN {X 19.135,Y 97.1147,Z 97,A 74.0686,B 24.9153,C -2.1248,E1 25.0304,E2 371.2155} C_DIS
LIN {X 16.4429,Y 97.6057,Z 97,A 75.8989,B 24.9146,C -2.1344,E1 25.0254,E2 369.3642} C_DIS
LIN {X 12.8293,Y 98.146,Z 97,A 77.9445,B 24.9147,C -2.1324,E1 25.0197,E2 367.3252} C_DIS
LIN {X 9.9045,Y 98.4849,Z 97,A 79.7215,B 24.9145,C -2.1353,E1 25.0148,E2 365.5425} C_DIS
LIN {X 6.5143,Y 98.7665,Z 97,A 82.3,B 24.9127,C -2.1578,E1 25.0074,E2 362.9118} C_DIS
LIN {X 2.3736,Y 98.9537,Z 97,A 83.8753,B 24.9151,C -2.1274,E1 25.0033,E2 361.409} C_DIS
LIN {X -4.1885,Y 98.8923,Z 97,A 87.4611,B 24.9158,C -2.1187,E1 24.9933,E2 357.8437} C_DIS
LIN {X -9.7311,Y 98.5031,Z 97,A 91.0578,B 24.9148,C -2.1309,E1 24.9832,E2 354.2167} C_DIS
LIN {X -13.026,Y 98.1205,Z 97,A 92.8914,B 24.9152,C -2.1267,E1 24.9781,E2 352.3918} C_DIS
LIN {X -16.3371,Y 97.6234,Z 97,A 94.9187,B 24.915,C -2.1285,E1 24.9725,E2 350.3582} C_DIS
LIN {X -19.8101,Y 96.9783,Z 97,A 97.049,B 24.915,C -2.1299,E1 24.9667,E2 348.2222} C_DIS
LIN {X -23.7389,Y 96.0925,Z 97,A 99.3113,B 24.9153,C -2.1253,E1 24.9605,E2 345.9679} C_DIS
LIN {X -28.6318,Y 94.7507,Z 97,A 102.9174,B 24.9136,C -2.1459,E1 24.9507,E2 342.3069} C_DIS
LIN {X -32.4929,Y 93.4961,Z 97,A 104.3377,B 24.9165,C -2.1102,E1 24.9472,E2 340.9689} C_DIS
LIN {X -37.0833,Y 91.7721,Z 97,A 107.4295,B 24.9161,C -2.1152,E1 24.9391,E2 337.8586} C_DIS
LIN {X -39.9902,Y 90.5441,Z 97,A 109.3165,B 24.9161,C -2.1147,E1 24.9342,E2 335.9684} C_DIS
LIN {X -43.0464,Y 89.1306,Z 97,A 111.1517,B 24.9167,C -2.1077,E1 24.9296,E2 334.1453} C_DIS
LIN {X -45.7396,Y 87.7798,Z 97,A 113.0435,B 24.9165,C -2.11,E1 24.9249,E2 332.2429} C_DIS
LIN {X -52.1486,Y 84.13,Z 97,A 117.2886,B 24.9172,C -2.1014,E1 24.9147,E2 328.0054} C_DIS
LIN {X -54.2611,Y 82.783,Z 97,A 119.2553,B 24.916,C -2.1165,E1 24.91,E2 325.9963} C_DIS
LIN {X -57.2012,Y 80.7798,Z 97,A 120.5656,B 24.9184,C -2.0865,E1 24.9071,E2 324.753} C_DIS
LIN {X -59.2366,Y 79.2989,Z 97,A 122.3357,B 24.9177,C -2.0943,E1 24.9031,E2 322.9582} C_DIS
LIN {X -62.2253,Y 76.9756,Z 97,A 124.4687,B 24.9183,C -2.0876,E1 24.8984,E2 320.8333} C_DIS
LIN {X -65.4216,Y 74.2791,Z 97,A 127.0697,B 24.9183,C -2.0883,E1 24.8929,E2 318.2204} C_DIS
LIN {X -68.4007,Y 71.5453,Z 97,A 129.3378,B 24.9188,C -2.0803,E1 24.8883,E2 315.962} C_DIS
LIN {X -70.8912,Y 69.0793,Z 97,A 131.2889,B 24.9194,C -2.0728,E1 24.8845,E2 314.0206} C_DIS
LIN {X -73.5811,Y 66.2051,Z 97,A 134.2209,B 24.9181,C -2.0893,E1 24.8789,E2 311.0361} C_DIS
LIN {X -76.1675,Y 63.2118,Z 97,A 135.7335,B 24.9207,C -2.057,E1 24.8763,E2 309.5937} C_DIS
LIN {X -78.0193,Y 60.9143,Z 97,A 137.7249,B 24.9203,C -2.062,E1 24.8728,E2 307.5809} C_DIS
LIN {X -80.1302,Y 58.1083,Z 97,A 140.4698,B 24.9188,C -2.0807,E1 24.8682,E2 304.7781} C_DIS
LIN {X -82.7528,Y 54.3069,Z 97,A 142.2454,B 24.9217,C -2.0428,E1 24.8656,E2 303.084} C_DIS
LIN {X -84.3545,Y 51.7854,Z 97,A 143.892,B 24.9223,C -2.0352,E1 24.8632,E2 301.4473} C_DIS
LIN {X -86.3007,Y 48.4713,Z 97,A 146.3303,B 24.9223,C -2.0359,E1 24.8597,E2 298.9945} C_DIS
LIN {X -87.8029,Y 45.6958,Z 97,A 148.3668,B 24.9221,C -2.0376,E1 24.8571,E2 296.9432} C_DIS
LIN {X -89.6678,Y 41.9157,Z 97,A 150.6109,B 24.9232,C -2.0238,E1 24.8544,E2 294.72} C_DIS
LIN {X -91.0624,Y 38.7945,Z 97,A 152.6087,B 24.9236,C -2.0184,E1 24.8521,E2 292.7239} C_DIS
LIN {X -92.2509,Y 35.8764,Z 97,A 154.4284,B 24.924,C -2.0127,E1 24.8503,E2 290.9077} C_DIS
LIN {X -93.5009,Y 32.4793,Z 97,A 156.4704,B 24.9247,C -2.0044,E1 24.8483,E2 288.8738} C_DIS
LIN {X -94.7203,Y 28.7331,Z 97,A 158.7102,B 24.9253,C -1.9959,E1 24.8464,E2 286.6414} C_DIS
LIN {X -95.66,Y 25.4274,Z 97,A 160.742,B 24.9257,C -1.9911,E1 24.8449,E2 284.6094} C_DIS
LIN {X -96.3586,Y 22.6357,Z 97,A 162.5831,B 24.9257,C -1.9916,E1 24.8437,E2 282.7562} C_DIS
LIN {X -97.0961,Y 19.2312,Z 97,A 164.7045,B 24.9258,C -1.9887,E1 24.8425,E2 280.6293} C_DIS
LIN {X -97.598,Y 16.4888,Z 97,A 166.2865,B 24.9263,C -1.9825,E1 24.8418,E2 279.0528} C_DIS
LIN {X -98.147,Y 12.8221,Z 97,A 168.3148,B 24.9271,C -1.9717,E1 24.841,E2 277.0382} C_DIS
LIN {X -98.503,Y 9.7321,Z 97,A 170.2607,B 24.9271,C -1.9707,E1 24.8404,E2 275.0829} C_DIS
LIN {X -98.7909,Y 6.1529,Z 97,A 172.2568,B 24.9279,C -1.9612,E1 24.84,E2 273.0973} C_DIS
LIN {X -98.9403,Y 2.8427,Z 97,A 174.0411,B 24.9287,C -1.9506,E1 24.8398,E2 271.3276} C_DIS
LIN {X -98.983,Y -0.1014,Z 97,A 175.7906,B 24.929,C -1.9466,E1 24.8398,E2 269.5771} C_DIS
LIN {X -98.9574,Y -2.1869,Z 97,A 177.1819,B 24.9288,C -1.9489,E1 24.8398,E2 268.172} C_DIS
LIN {X -98.8394,Y -5.2935,Z 97,A 179.0106,B 24.9291,C -1.9441,E1 24.8401,E2 266.3437} C_DIS
LIN {X -98.6306,Y -8.3322,Z 97,A -179.1844,B 24.9294,C -1.9399,E1 24.8405,E2 264.538} C_DIS
LIN {X -98.2375,Y -12.1237,Z 97,A -177.1277,B 24.9303,C -1.9279,E1 24.8411,E2 262.4976} C_DIS
LIN {X -97.768,Y -15.4516,Z 97,A -175.0507,B 24.9304,C -1.9262,E1 24.842,E2 260.4123} C_DIS
LIN {X -97.2409,Y -18.4795,Z 97,A -173.0018,B 24.9302,C -1.9297,E1 24.8431,E2 258.3428} C_DIS
LIN {X -96.3201,Y -22.8024,Z 97,A -170.6313,B 24.9312,C -1.9155,E1 24.8445,E2 255.9924} C_DIS
LIN {X -95.4883,Y -26.0628,Z 97,A -168.7525,B 24.9318,C -1.9072,E1 24.8459,E2 254.1223} C_DIS
LIN {X -94.409,Y -29.7383,Z 97,A -166.0567,B 24.9311,C -1.9167,E1 24.8481,E2 251.3884} C_DIS
LIN {X -93.3301,Y -32.9661,Z 97,A -164.7499,B 24.9331,C -1.8884,E1 24.8493,E2 250.1416} C_DIS
LIN {X -92.4521,Y -35.3545,Z 97,A -163.0166,B 24.9328,C -1.8929,E1 24.851,E2 248.3879} C_DIS
LIN {X -91.2545,Y -38.3386,Z 97,A -161.2365,B 24.9334,C -1.8848,E1 24.8528,E2 246.6173} C_DIS
LIN {X -90.0678,Y -41.0511,Z 97,A -159.3734,B 24.9334,C -1.8849,E1 24.855,E2 244.7435} C_DIS
LIN {X -88.7306,Y -43.8648,Z 97,A -156.6794,B 24.9316,C -1.9105,E1 24.8585,E2 241.9742} C_DIS
LIN {X -86.2357,Y -48.5878,Z 97,A -154.7268,B 24.9349,C -1.863,E1 24.8609,E2 240.1245} C_DIS
LIN {X -84.7326,Y -51.1634,Z 97,A -152.8772,B 24.9349,C -1.8626,E1 24.8636,E2 238.2663} C_DIS
LIN {X -83.1091,Y -53.7607,Z 97,A -151.1502,B 24.9354,C -1.8564,E1 24.8661,E2 236.5452} C_DIS
LIN {X -81.6985,Y -55.8819,Z 97,A -149.5301,B 24.9354,C -1.8576,E1 24.8687,E2 234.9142} C_DIS
LIN {X -79.6011,Y -58.831,Z 97,A -147.3668,B 24.9355,C -1.8548,E1 24.8723,E2 232.747} C_DIS
LIN {X -77.4869,Y -61.5879,Z 97,A -145.515,B 24.9362,C -1.8445,E1 24.8754,E2 230.911} C_DIS
LIN {X -75.2923,Y -64.2518,Z 97,A -143.3873,B 24.9362,C -1.8444,E1 24.8792,E2 228.7739} C_DIS
LIN {X -72.851,Y -67.0072,Z 97,A -141.3319,B 24.9367,C -1.837,E1 24.8831,E2 226.7269} C_DIS
LIN {X -70.5624,Y -69.4133,Z 97,A -139.3962,B 24.937,C -1.8333,E1 24.8868,E2 224.7917} C_DIS
LIN {X -68.4435,Y -71.5041,Z 97,A -137.4821,B 24.9368,C -1.8364,E1 24.8907,E2 222.8623} C_DIS
LIN {X -65.6621,Y -74.0672,Z 97,A -135.3164,B 24.9371,C -1.8312,E1 24.8952,E2 220.7003} C_DIS
LIN {X -62.8796,Y -76.4436,Z 97,A -133.3602,B 24.9378,C -1.8215,E1 24.8993,E2 218.7596} C_DIS
LIN {X -60.1395,Y -78.6167,Z 97,A -131.3129,B 24.938,C -1.8186,E1 24.9038,E2 216.7116} C_DIS
LIN {X -56.0361,Y -81.5935,Z 97,A -128.4357,B 24.9385,C -1.8116,E1 24.9104,E2 213.841} C_DIS
LIN {X -53.9113,Y -83.0125,Z 97,A -126.7974,B 24.9383,C -1.8149,E1 24.9142,E2 212.1895} C_DIS
LIN {X -50.9162,Y -84.8828,Z 97,A -124.5763,B 24.938,C -1.8182,E1 24.9195,E2 209.9538} C_DIS
LIN {X -47.7643,Y -86.6955,Z 97,A -122.778,B 24.939,C -1.8044,E1 24.9238,E2 208.1831} C_DIS
LIN {X -45.2945,Y -88.0097,Z 97,A -120.5428,B 24.9376,C -1.8244,E1 24.9295,E2 205.8942} C_DIS
LIN {X -42.1409,Y -89.563,Z 97,A -119.2152,B 24.9395,C -1.7966,E1 24.9327,E2 204.6294} C_DIS
LIN {X -38.1888,Y -91.3176,Z 97,A -116.4752,B 24.9391,C -1.8024,E1 24.9398,E2 201.869} C_DIS
LIN {X -34.7993,Y -92.6623,Z 97,A -114.6262,B 24.9399,C -1.791,E1 24.9445,E2 200.0433} C_DIS
LIN {X -32.5198,Y -93.4867,Z 97,A -113.0689,B 24.9396,C -1.7953,E1 24.9487,E2 198.4726} C_DIS
LIN {X -29.41,Y -94.5107,Z 97,A -111.0207,B 24.9393,C -1.7994,E1 24.9541,E2 196.411} C_DIS
LIN {X -26.3096,Y -95.4217,Z 97,A -109.1381,B 24.9393,C -1.7986,E1 24.9592,E2 194.5273} C_DIS
LIN {X -23.2692,Y -96.2071,Z 97,A -107.4066,B 24.9396,C -1.7945,E1 24.9639,E2 192.8032} C_DIS
LIN {X -19.8676,Y -96.9665,Z 97,A -104.7928,B 24.9382,C -1.8155,E1 24.9712,E2 190.1362} C_DIS
LIN {X -16.1743,Y -97.6506,Z 97,A -102.6593,B 24.9384,C -1.8134,E1 24.977,E2 188.0059} C_DIS
LIN {X -12.6245,Y -98.1726,Z 97,A -101.2172,B 24.94,C -1.7894,E1 24.9809,E2 186.6195} C_DIS
LIN {X -10.4548,Y -98.4273,Z 97,A -99.1888,B 24.9381,C -1.8177,E1 24.9867,E2 184.5229} C_DIS
LIN {X -6.3821,Y -98.7754,Z 97,A -97.5781,B 24.94,C -1.7895,E1 24.991,E2 182.9784} C_DIS
LIN {X -1.8738,Y -98.9632,Z 97,A -94.903,B 24.9398,C -1.7922,E1 24.9985,E2 180.2965} C_DIS
LIN {X 0.6835,Y -98.9739,Z 97,A -93.8445,B 24.9408,C -1.7769,E1 25.0013,E2 179.2743} C_DIS
Enddeposition()
LIN {X 0.6835,Y -98.9739,Z 97,A -93.8445,B 24.9408,C -1.7769,E1 25.0013,E2 179.2743} C_DIS
Startdeposition()
$VEL.CP = VEL_PRINT
LIN {X -4.7496,Y -97.9628,Z 97,A -98.2779,B 24.9428,C -1.7467,E1 24.9888,E2 183.7801} C_DIS
LIN {X -9.3814,Y -97.6274,Z 97,A -100.2522,B 24.9411,C -1.7732,E1 24.9835,E2 185.6923} C_DIS
LIN {X -14.2572,Y -97.0346,Z 97,A -103.194,B 24.9412,C -1.7712,E1 24.9753,E2 188.6411} C_DIS
LIN {X -19.0463,Y -96.2106,Z 97,A -105.9577,B 24.941,C -1.7749,E1 24.9677,E2 191.399} C_DIS
LIN {X -21.7294,Y -95.6397,Z 97,A -107.6723,B 24.9412,C -1.7717,E1 24.963,E2 193.1234} C_DIS
LIN {X -25.5922,Y -94.6785,Z 97,A -109.7927,B 24.9406,C -1.7803,E1 24.9573,E2 195.2264} C_DIS
LIN {X -28.8552,Y -93.7358,Z 97,A -111.7203,B 24.9404,C -1.7837,E1 24.9522,E2 197.1492} C_DIS
LIN {X -31.7889,Y -92.783,Z 97,A -113.7297,B 24.9408,C -1.7778,E1 24.9468,E2 199.1763} C_DIS
LIN {X -37.3977,Y -90.6676,Z 97,A -117.9807,B 24.9423,C -1.7552,E1 24.9356,E2 203.4902} C_DIS
LIN {X -41.8152,Y -88.7169,Z 97,A -120.2606,B 24.9408,C -1.7771,E1 24.93,E2 205.7238} C_DIS
LIN {X -45.6556,Y -86.8018,Z 97,A -122.5069,B 24.94,C -1.7893,E1 24.9244,E2 207.9472} C_DIS
LIN {X -48.2831,Y -85.3699,Z 97,A -124.9958,B 24.9415,C -1.7663,E1 24.9182,E2 210.4981} C_DIS
LIN {X -52.1221,Y -83.0802,Z 97,A -127.3397,B 24.9407,C -1.7793,E1 24.9127,E2 212.8184} C_DIS
LIN {X -55.0488,Y -81.1703,Z 97,A -129.4669,B 24.9407,C -1.7797,E1 24.9078,E2 214.9517} C_DIS
LIN {X -58.1609,Y -78.9707,Z 97,A -131.119,B 24.9391,C -1.8031,E1 24.9042,E2 216.5541} C_DIS
LIN {X -61.4527,Y -76.4375,Z 97,A -133.6196,B 24.9389,C -1.8049,E1 24.8987,E2 219.0595} C_DIS
LIN {X -65.0169,Y -73.4307,Z 97,A -136.3278,B 24.9385,C -1.8107,E1 24.8929,E2 221.7645} C_DIS
LIN {X -68.9151,Y -69.7832,Z 97,A -139.4089,B 24.938,C -1.8184,E1 24.8867,E2 224.84} C_DIS
LIN {X -71.4089,Y -67.2291,Z 97,A -141.5105,B 24.9378,C -1.8223,E1 24.8827,E2 226.9412} C_DIS
LIN {X -73.2918,Y -65.1721,Z 97,A -143.5969,B 24.9385,C -1.8107,E1 24.8787,E2 229.0647} C_DIS
LIN {X -75.3979,Y -62.7228,Z 97,A -145.0022,B 24.9371,C -1.8311,E1 24.8763,E2 230.4277} C_DIS
LIN {X -76.7742,Y -61.031,Z 97,A -146.5405,B 24.9375,C -1.8253,E1 24.8735,E2 231.987} C_DIS
LIN {X -79.1572,Y -57.9062,Z 97,A -149.0289,B 24.9375,C -1.8246,E1 24.8694,E2 234.4893} C_DIS
LIN {X -81.8796,Y -53.9881,Z 97,A -151.436,B 24.9362,C -1.8442,E1 24.8657,E2 236.8615} C_DIS
LIN {X -83.6082,Y -51.272,Z 97,A -153.37,B 24.936,C -1.8474,E1 24.8628,E2 238.7979} C_DIS
LIN {X -85.3796,Y -48.2656,Z 97,A -155.3819,B 24.9356,C -1.8537,E1 24.86,E2 240.8052} C_DIS
LIN {X -87.8988,Y -43.5062,Z 97,A -158.1954,B 24.9342,C -1.8733,E1 24.8564,E2 243.5868} C_DIS
LIN {X -89.1475,Y -40.8902,Z 97,A -160.318,B 24.9349,C -1.8639,E1 24.8538,E2 245.7435} C_DIS
LIN {X -90.559,Y -37.6599,Z 97,A -162.3261,B 24.9343,C -1.8715,E1 24.8516,E2 247.7445} C_DIS
LIN {X -91.7441,Y -34.6701,Z 97,A -164.205,B 24.934,C -1.877,E1 24.8497,E2 249.6209} C_DIS
LIN {X -92.6118,Y -32.2812,Z 97,A -166.0212,B 24.9344,C -1.8706,E1 24.848,E2 251.4628} C_DIS
LIN {X -94.7995,Y -25.1446,Z 97,A -170.182,B 24.933,C -1.8902,E1 24.8448,E2 255.6006} C_DIS
LIN {X -96.3112,Y -18.5242,Z 97,A -173.9644,B 24.9317,C -1.9085,E1 24.8425,E2 259.3616} C_DIS
LIN {X -96.8791,Y -15.2811,Z 97,A -176.0527,B 24.9317,C -1.9092,E1 24.8415,E2 261.4609} C_DIS
LIN {X -97.3388,Y -12.02,Z 97,A -178.0875,B 24.9315,C -1.9116,E1 24.8408,E2 263.5019} C_DIS
LIN {X -97.7384,Y -8.1429,Z 97,A 179.7036,B 24.9308,C -1.9211,E1 24.8402,E2 265.7015} C_DIS
LIN {X -97.9754,Y -4.4578,Z 97,A 177.5584,B 24.9303,C -1.9284,E1 24.8399,E2 267.8423} C_DIS
LIN {X -98.0704,Y -1.2285,Z 97,A 175.6407,B 24.9299,C -1.9334,E1 24.8398,E2 269.7594} C_DIS
LIN {X -98.0562,Y 2.0042,Z 97,A 173.6246,B 24.9298,C -1.9354,E1 24.8398,E2 271.783} C_DIS
LIN {X -97.9529,Y 4.9427,Z 97,A 171.8913,B 24.9294,C -1.9404,E1 24.8401,E2 273.5147} C_DIS
LIN {X -97.6813,Y 8.7971,Z 97,A 169.6681,B 24.9288,C -1.9488,E1 24.8406,E2 275.7313} C_DIS
LIN {X -97.271,Y 12.5435,Z 97,A 167.4882,B 24.9282,C -1.9566,E1 24.8413,E2 277.9057} C_DIS
LIN {X -96.8366,Y 15.5563,Z 97,A 165.7441,B 24.9277,C -1.9633,E1 24.842,E2 279.644} C_DIS
LIN {X -95.9764,Y 20.1929,Z 97,A 162.9067,B 24.9273,C -1.9695,E1 24.8435,E2 282.4835} C_DIS
LIN {X -95.2611,Y 23.3308,Z 97,A 161.142,B 24.9266,C -1.9792,E1 24.8447,E2 284.2354} C_DIS
LIN {X -94.5854,Y 25.937,Z 97,A 159.6809,B 24.9259,C -1.9878,E1 24.8457,E2 285.6845} C_DIS
LIN {X -93.3818,Y 29.9813,Z 97,A 157.0505,B 24.9257,C -1.9901,E1 24.8479,E2 288.3245} C_DIS
LIN {X -92.6619,Y 32.1386,Z 97,A 155.0209,B 24.9271,C -1.9717,E1 24.8498,E2 290.4096} C_DIS
LIN {X -91.2693,Y 35.9012,Z 97,A 153.3022,B 24.9251,C -1.999,E1 24.8515,E2 292.0729} C_DIS
LIN {X -89.9905,Y 38.9966,Z 97,A 151.3032,B 24.9247,C -2.0035,E1 24.8536,E2 294.072} C_DIS
LIN {X -88.4905,Y 42.2902,Z 97,A 148.7112,B 24.9254,C -1.9944,E1 24.8568,E2 296.6999} C_DIS
LIN {X -86.9198,Y 45.4316,Z 97,A 147.4293,B 24.9231,C -2.0254,E1 24.8583,E2 297.9147} C_DIS
LIN {X -84.2031,Y 50.2893,Z 97,A 144.0098,B 24.9228,C -2.0293,E1 24.863,E2 301.3428} C_DIS
LIN {X -82.2916,Y 53.3599,Z 97,A 141.8925,B 24.9223,C -2.0351,E1 24.8662,E2 303.457} C_DIS
LIN {X -78.1777,Y 59.2233,Z 97,A 137.6315,B 24.9217,C -2.044,E1 24.8731,E2 307.7177} C_DIS
LIN {X -74.8877,Y 63.3315,Z 97,A 134.5155,B 24.9211,C -2.0507,E1 24.8785,E2 310.8323} C_DIS
LIN {X -70.4789,Y 68.2037,Z 97,A 130.4927,B 24.9209,C -2.0542,E1 24.8862,E2 314.8644} C_DIS
LIN {X -66.5597,Y 72.0341,Z 97,A 127.6123,B 24.9195,C -2.0724,E1 24.8919,E2 317.7133} C_DIS
LIN {X -62.3026,Y 75.7471,Z 97,A 124.2789,B 24.919,C -2.0787,E1 24.8989,E2 321.0449} C_DIS
LIN {X -59.5207,Y 77.9495,Z 97,A 121.7943,B 24.9197,C -2.0694,E1 24.9044,E2 323.5607} C_DIS
LIN {X -56.1908,Y 80.3839,Z 97,A 119.4514,B 24.9191,C -2.0765,E1 24.9097,E2 325.8949} C_DIS
LIN {X -52.8221,Y 82.6369,Z 97,A 116.6992,B 24.9198,C -2.0682,E1 24.9163,E2 328.6757} C_DIS
LIN {X -49.9463,Y 84.4059,Z 97,A 114.8214,B 24.9193,C -2.075,E1 24.9207,E2 330.5432} C_DIS
LIN {X -46.5874,Y 86.3055,Z 97,A 112.4285,B 24.9193,C -2.0742,E1 24.9266,E2 332.9448} C_DIS
LIN {X -43.4988,Y 87.9025,Z 97,A 110.9393,B 24.9176,C -2.0957,E1 24.9302,E2 334.3867} C_DIS
LIN {X -40.4465,Y 89.3482,Z 97,A 108.9238,B 24.9176,C -2.0973,E1 24.9353,E2 336.4036} C_DIS
LIN {X -37.0768,Y 90.7982,Z 97,A 106.5009,B 24.918,C -2.0908,E1 24.9416,E2 338.8473} C_DIS
LIN {X -32.9074,Y 92.3921,Z 97,A 104.0591,B 24.9173,C -2.0998,E1 24.948,E2 341.2726} C_DIS
LIN {X -28.3747,Y 93.8835,Z 97,A 101.2221,B 24.9172,C -2.1014,E1 24.9555,E2 344.111} C_DIS
LIN {X -23.5425,Y 95.2094,Z 97,A 98.4209,B 24.9166,C -2.1087,E1 24.9631,E2 346.899} C_DIS
LIN {X -20.4766,Y 95.916,Z 97,A 96.4828,B 24.9168,C -2.1068,E1 24.9684,E2 348.8439} C_DIS
LIN {X -17.4783,Y 96.5065,Z 97,A 94.6627,B 24.9168,C -2.107,E1 24.9734,E2 350.6656} C_DIS
LIN {X -13.7545,Y 97.1072,Z 97,A 92.6381,B 24.9161,C -2.1148,E1 24.9789,E2 352.6735} C_DIS
LIN {X -10.0165,Y 97.5638,Z 97,A 89.9919,B 24.9173,C -2.1004,E1 24.9864,E2 355.3555} C_DIS
LIN {X -4.9723,Y 97.9513,Z 97,A 87.4715,B 24.916,C -2.1168,E1 24.9933,E2 357.8378} C_DIS
LIN {X 1.5682,Y 98.0642,Z 97,A 83.6396,B 24.916,C -2.1173,E1 25.004,E2 361.6686} C_DIS
LIN {X 5.9457,Y 97.8975,Z 97,A 80.937,B 24.9163,C -2.1123,E1 25.0115,E2 364.3822} C_DIS
LIN {X 9.4583,Y 97.6203,Z 97,A 78.9165,B 24.9163,C -2.1135,E1 25.0171,E2 366.3987} C_DIS
LIN {X 13.12,Y 97.1963,Z 97,A 76.8069,B 24.9161,C -2.1146,E1 25.023,E2 368.504} C_DIS
LIN {X 16.3029,Y 96.712,Z 97,A 74.928,B 24.9161,C -2.1141,E1 25.0282,E2 370.3823} C_DIS
LIN {X 18.7829,Y 96.2614,Z 97,A 73.2465,B 24.9168,C -2.106,E1 25.0328,E2 372.0811} C_DIS
LIN {X 22.9784,Y 95.347,Z 97,A 70.9565,B 24.9163,C -2.1125,E1 25.039,E2 374.3523} C_DIS
LIN {X 26.1836,Y 94.5183,Z 97,A 69.0346,B 24.9163,C -2.1117,E1 25.0442,E2 376.2732} C_DIS
LIN {X 28.8905,Y 93.7249,Z 97,A 67.4052,B 24.9164,C -2.1112,E1 25.0485,E2 377.901} C_DIS
LIN {X 34.0128,Y 91.9908,Z 97,A 64.3562,B 24.9164,C -2.1125,E1 25.0566,E2 380.9408} C_DIS
LIN {X 40.7612,Y 89.2064,Z 97,A 59.9044,B 24.9172,C -2.101,E1 25.0681,E2 385.4093} C_DIS
LIN {X 44.2577,Y 87.5238,Z 97,A 57.9337,B 24.9166,C -2.1092,E1 25.0729,E2 387.3555} C_DIS
LIN {X 48.2785,Y 85.3724,Z 97,A 55.0106,B 24.9176,C -2.0959,E1 25.0802,E2 390.3016} C_DIS
LIN {X 51.5877,Y 83.414,Z 97,A 51.9003,B 24.9204,C -2.0606,E1 25.0877,E2 393.4855} C_DIS
LIN {X 55.8126,Y 80.6473,Z 97,A 50.005,B 24.9177,C -2.0949,E1 25.0919,E2 395.2934} C_DIS
LIN {X 58.8316,Y 78.4719,Z 97,A 47.7752,B 24.9182,C -2.089,E1 25.0969,E2 397.5291} C_DIS
LIN {X 61.2754,Y 76.5808,Z 97,A 45.8126,B 24.9189,C -2.0798,E1 25.1013,E2 399.5063} C_DIS
LIN {X 65.1979,Y 73.2687,Z 97,A 42.7503,B 24.9195,C -2.0716,E1 25.1078,E2 402.576} C_DIS
LIN {X 68.8221,Y 69.875,Z 97,A 40.0999,B 24.9193,C -2.075,E1 25.1131,E2 405.2072} C_DIS
LIN {X 70.9068,Y 67.7598,Z 97,A 38.4214,B 24.9193,C -2.0734,E1 25.1164,E2 406.8824} C_DIS
LIN {X 73.437,Y 65.01,Z 97,A 36.1993,B 24.9199,C -2.067,E1 25.1205,E2 409.1097} C_DIS
LIN {X 75.3844,Y 62.739,Z 97,A 34.3769,B 24.9204,C -2.0601,E1 25.1238,E2 410.9401} C_DIS
LIN {X 78.0965,Y 59.3311,Z 97,A 31.8684,B 24.9208,C -2.0554,E1 25.1281,E2 413.4481} C_DIS
LIN {X 79.9842,Y 56.759,Z 97,A 29.9411,B 24.9213,C -2.0483,E1 25.1313,E2 415.3827} C_DIS
LIN {X 83.2887,Y 51.7883,Z 97,A 26.4734,B 24.922,C -2.04,E1 25.1366,E2 418.8526} C_DIS
LIN {X 84.9427,Y 49.0282,Z 97,A 24.0357,B 24.924,C -2.0136,E1 25.1401,E2 421.3402} C_DIS
LIN {X 86.9078,Y 45.4543,Z 97,A 22.2681,B 24.9227,C -2.0307,E1 25.1423,E2 423.0581} C_DIS
LIN {X 88.7347,Y 41.777,Z 97,A 18.8803,B 24.9261,C -1.9859,E1 25.1465,E2 426.5332} C_DIS
LIN {X 90.9577,Y 36.6848,Z 97,A 16.6206,B 24.9239,C -2.0145,E1 25.1488,E2 428.7132} C_DIS
LIN {X 91.9452,Y 34.1378,Z 97,A 14.2781,B 24.9264,C -1.9809,E1 25.1512,E2 431.1218} C_DIS
LIN {X 93.5033,Y 29.6048,Z 97,A 12.1337,B 24.9252,C -1.9978,E1 25.1529,E2 433.2141} C_DIS
LIN {X 94.6724,Y 25.6148,Z 97,A 9.9057,B 24.9252,C -1.9983,E1 25.1546,E2 435.4282} C_DIS
LIN {X 95.5057,Y 22.3092,Z 97,A 7.8203,B 24.9259,C -1.9885,E1 25.156,E2 437.5247} C_DIS
LIN {X 96.3311,Y 18.4206,Z 97,A 5.6429,B 24.9259,C -1.9869,E1 25.1572,E2 439.6931} C_DIS
LIN {X 96.9447,Y 14.8568,Z 97,A 3.4968,B 24.9266,C -1.979,E1 25.1582,E2 441.8453} C_DIS
LIN {X 97.434,Y 11.2088,Z 97,A 1.3216,B 24.9271,C -1.9712,E1 25.1589,E2 444.0261} C_DIS
LIN {X 97.7686,Y 7.7641,Z 97,A -0.901,B 24.9282,C -1.9569,E1 25.1594,E2 446.2692} C_DIS
LIN {X 98.0128,Y 3.5773,Z 97,A -4.1351,B 24.931,C -1.9186,E1 25.1598,E2 449.5745} C_DIS
LIN {X 98.0536,Y -2.1427,Z 97,A -6.3561,B 24.9286,C -1.9514,E1 25.1598,E2 451.7048} C_DIS
LIN {X 97.7227,Y -8.3355,Z 97,A -10.2951,B 24.9304,C -1.9273,E1 25.159,E2 455.6773} C_DIS
LIN {X 97.2505,Y -12.7016,Z 97,A -12.373,B 24.9296,C -1.9382,E1 25.1583,E2 457.7171} C_DIS
LIN {X 96.8157,Y -15.683,Z 97,A -14.3236,B 24.9305,C -1.925,E1 25.1575,E2 459.6874} C_DIS
LIN {X 96.3501,Y -18.3221,Z 97,A -15.8217,B 24.9307,C -1.9227,E1 25.1567,E2 461.1823} C_DIS
LIN {X 95.632,Y -21.7625,Z 97,A -17.9374,B 24.9313,C -1.9137,E1 25.1555,E2 463.3069} C_DIS
LIN {X 94.8007,Y -25.1398,Z 97,A -19.8012,B 24.9313,C -1.9138,E1 25.1542,E2 465.1597} C_DIS
LIN {X 93.4406,Y -29.7996,Z 97,A -22.7344,B 24.9322,C -1.9011,E1 25.1518,E2 468.1061} C_DIS
LIN {X 92.6365,Y -32.2111,Z 97,A -24.105,B 24.9322,C -1.9009,E1 25.1506,E2 469.4694} C_DIS
LIN {X 91.0946,Y -36.3458,Z 97,A -26.5841,B 24.9325,C -1.8968,E1 25.1481,E2 471.9443} C_DIS
LIN {X 90.2374,Y -38.4232,Z 97,A -28.5308,B 24.9346,C -1.8681,E1 25.1459,E2 473.9482} C_DIS
LIN {X 88.7835,Y -41.6722,Z 97,A -29.8048,B 24.9328,C -1.8933,E1 25.1445,E2 475.1558} C_DIS
LIN {X 87.5455,Y -44.2154,Z 97,A -31.535,B 24.9334,C -1.8853,E1 25.1424,E2 476.8957} C_DIS
LIN {X 84.3555,Y -50.0316,Z 97,A -35.579,B 24.9346,C -1.8673,E1 25.1369,E2 480.961} C_DIS
LIN {X 82.3899,Y -53.2069,Z 97,A -38.6219,B 24.9374,C -1.8278,E1 25.1322,E2 484.082} C_DIS
LIN {X 79.6032,Y -57.293,Z 97,A -40.8606,B 24.9362,C -1.8449,E1 25.1286,E2 486.2693} C_DIS
LIN {X 76.8658,Y -60.9151,Z 97,A -43.2024,B 24.9359,C -1.8498,E1 25.1247,E2 488.5884} C_DIS
LIN {X 74.7784,Y -63.4603,Z 97,A -45.0781,B 24.9361,C -1.8466,E1 25.1213,E2 490.463} C_DIS
LIN {X 72.3798,Y -66.1829,Z 97,A -47.4227,B 24.9371,C -1.8325,E1 25.1169,E2 492.8305} C_DIS
LIN {X 69.4933,Y -69.2086,Z 97,A -49.7595,B 24.9371,C -1.8306,E1 25.1124,E2 495.1618} C_DIS
LIN {X 67.0654,Y -71.5629,Z 97,A -51.7107,B 24.9374,C -1.8268,E1 25.1084,E2 497.1139} C_DIS
LIN {X 64.265,Y -74.0885,Z 97,A -54.1343,B 24.9384,C -1.8133,E1 25.1033,E2 499.5599} C_DIS
LIN {X 60.8782,Y -76.895,Z 97,A -56.4727,B 24.9382,C -1.8165,E1 25.0983,E2 501.8819} C_DIS
LIN {X 58.128,Y -78.9948,Z 97,A -58.4524,B 24.9383,C -1.8138,E1 25.0938,E2 503.8608} C_DIS
LIN {X 55.1261,Y -81.118,Z 97,A -61.0731,B 24.9398,C -1.7915,E1 25.0877,E2 506.5253} C_DIS
LIN {X 52.1669,Y -83.0522,Z 97,A -62.6131,B 24.9388,C -1.8074,E1 25.0842,E2 508.0226} C_DIS
LIN {X 49.2071,Y -84.8399,Z 97,A -64.4089,B 24.9384,C -1.8123,E1 25.0799,E2 509.8014} C_DIS
LIN {X 46.9628,Y -86.1019,Z 97,A -66.6969,B 24.9406,C -1.78,E1 25.0741,E2 512.1592} C_DIS
LIN {X 43.6582,Y -87.8235,Z 97,A -68.4025,B 24.9397,C -1.7941,E1 25.07,E2 513.8267} C_DIS
LIN {X 40.3193,Y -89.4055,Z 97,A -70.8679,B 24.9407,C -1.7792,E1 25.0636,E2 516.321} C_DIS
LIN {X 37.3561,Y -90.6844,Z 97,A -72.2255,B 24.9395,C -1.7963,E1 25.0603,E2 517.6351} C_DIS
LIN {X 34.7821,Y -91.7017,Z 97,A -74.6111,B 24.9416,C -1.7654,E1 25.0539,E2 520.0888} C_DIS
LIN {X 30.8436,Y -93.1017,Z 97,A -76.4103,B 24.9402,C -1.7862,E1 25.0492,E2 521.8351} C_DIS
LIN {X 27.7403,Y -94.0717,Z 97,A -78.0996,B 24.9398,C -1.7919,E1 25.0448,E2 523.5081} C_DIS
LIN {X 25.2751,Y -94.7642,Z 97,A -80.4126,B 24.9419,C -1.76,E1 25.0383,E2 525.8929} C_DIS
LIN {X 21.3312,Y -95.7296,Z 97,A -82.2006,B 24.9407,C -1.7792,E1 25.0336,E2 527.6328} C_DIS
LIN {X 17.8289,Y -96.4435,Z 97,A -84.233,B 24.9407,C -1.7795,E1 25.028,E2 529.6621} C_DIS
LIN {X 14.8812,Y -96.941,Z 97,A -86.0288,B 24.9409,C -1.7765,E1 25.0231,E2 531.4635} C_DIS
LIN {X 11.3525,Y -97.4172,Z 97,A -88.7547,B 24.9425,C -1.7516,E1 25.0154,E2 534.2462} C_DIS
LIN {X 7.0378,Y -97.8245,Z 97,A -90.3579,B 24.9403,C -1.7842,E1 25.0111,E2 535.7712} C_DIS
LIN {X 1.3262,Y -98.0686,Z 97,A -95.0999,B 24.9437,C -1.7325,E1 24.9975,E2 540.6349} C_DIS
LIN {X 1.3262,Y -98.0686,Z 97,A -95.0999,B 24.9437,C -1.7325,E1 24.9975,E2 540.6349} C_DIS
Enddeposition()
LIN {X 0.694,Y -97.1695,Z 97,A -93.9204,B 24.939,C -1.804,E1 25.0013,E2 539.2858} C_DIS
Startdeposition()
$VEL.CP = VEL_PRINT
LIN {X 6.0737,Y -96.9832,Z 97,A -90.2493,B 24.9377,C -1.8233,E1 25.0117,E2 535.5701} C_DIS
LIN {X 11.0377,Y -96.5434,Z 97,A -87.4506,B 24.9379,C -1.8197,E1 25.0194,E2 532.7816} C_DIS
LIN {X 13.7912,Y -96.1884,Z 97,A -85.6873,B 24.9375,C -1.8254,E1 25.0243,E2 531.0062} C_DIS
LIN {X 17.1363,Y -95.6491,Z 97,A -83.6817,B 24.9375,C -1.8273,E1 25.0299,E2 528.9983} C_DIS
LIN {X 20.8444,Y -94.9101,Z 97,A -81.4381,B 24.9372,C -1.8298,E1 25.036,E2 526.7516} C_DIS
LIN {X 26.089,Y -93.6052,Z 97,A -77.7034,B 24.9356,C -1.8537,E1 25.0462,E2 522.9661} C_DIS
LIN {X 29.6751,Y -92.5302,Z 97,A -76.1748,B 24.9372,C -1.8307,E1 25.0501,E2 521.4948} C_DIS
LIN {X 35.4625,Y -90.4699,Z 97,A -72.5187,B 24.9368,C -1.8367,E1 25.0598,E2 517.8321} C_DIS
LIN {X 38.8264,Y -89.0781,Z 97,A -70.4158,B 24.9367,C -1.8382,E1 25.0652,E2 515.7306} C_DIS
LIN {X 41.5471,Y -87.8441,Z 97,A -68.372,B 24.9357,C -1.8516,E1 25.0704,E2 513.6602} C_DIS
LIN {X 46.2834,Y -85.4415,Z 97,A -64.5434,B 24.9335,C -1.8839,E1 25.08,E2 509.7661} C_DIS
LIN {X 50.6206,Y -82.9456,Z 97,A -62.6364,B 24.9359,C -1.8491,E1 25.0844,E2 507.9474} C_DIS
LIN {X 55.0858,Y -80.0509,Z 97,A -59.0151,B 24.9342,C -1.8738,E1 25.0929,E2 504.2795} C_DIS
LIN {X 58.835,Y -77.338,Z 97,A -56.5813,B 24.9346,C -1.8682,E1 25.0983,E2 501.8679} C_DIS
LIN {X 61.325,Y -75.3769,Z 97,A -54.339,B 24.9333,C -1.8868,E1 25.1032,E2 499.5901} C_DIS
LIN {X 63.9062,Y -73.201,Z 97,A -52.5123,B 24.9333,C -1.885,E1 25.107,E2 497.7749} C_DIS
LIN {X 67.3587,Y -70.0372,Z 97,A -50.0889,B 24.9339,C -1.8783,E1 25.1119,E2 495.3771} C_DIS
LIN {X 69.7825,Y -67.623,Z 97,A -47.6732,B 24.9324,C -1.8989,E1 25.1167,E2 492.9232} C_DIS
LIN {X 71.9783,Y -65.2827,Z 97,A -45.6744,B 24.9318,C -1.9078,E1 25.1205,E2 490.9121} C_DIS
LIN {X 74.3207,Y -62.6029,Z 97,A -44.265,B 24.9333,C -1.8863,E1 25.123,E2 489.56} C_DIS
LIN {X 76.9575,Y -59.329,Z 97,A -41.0351,B 24.9307,C -1.9224,E1 25.1286,E2 486.2599} C_DIS
LIN {X 79.287,Y -56.1789,Z 97,A -39.2429,B 24.9317,C -1.9083,E1 25.1315,E2 484.5097} C_DIS
LIN {X 81.6228,Y -52.7274,Z 97,A -36.9268,B 24.9317,C -1.9097,E1 25.135,E2 482.2019} C_DIS
LIN {X 83.1709,Y -50.25,Z 97,A -34.0192,B 24.9279,C -1.9616,E1 25.1394,E2 479.1866} C_DIS
LIN {X 86.1099,Y -45.0284,Z 97,A -32.0073,B 24.9315,C -1.9117,E1 25.1419,E2 477.3032} C_DIS
LIN {X 87.8378,Y -41.5603,Z 97,A -29.29,B 24.9298,C -1.9355,E1 25.1453,E2 474.5443} C_DIS
LIN {X 89.6337,Y -37.5265,Z 97,A -26.6932,B 24.9292,C -1.9432,E1 25.1481,E2 471.9435} C_DIS
LIN {X 92.0296,Y -31.1925,Z 97,A -23.0842,B 24.9294,C -1.9403,E1 25.1516,E2 468.3614} C_DIS
LIN {X 93.5822,Y -26.1701,Z 97,A -19.6591,B 24.9278,C -1.9629,E1 25.1544,E2 464.9027} C_DIS
LIN {X 94.3282,Y -23.3382,Z 97,A -18.1132,B 24.9278,C -1.9612,E1 25.1554,E2 463.3696} C_DIS
LIN {X 95.0626,Y -20.143,Z 97,A -16.1927,B 24.9275,C -1.9668,E1 25.1566,E2 461.447} C_DIS
LIN {X 95.7361,Y -16.6524,Z 97,A -13.8576,B 24.9263,C -1.983,E1 25.1578,E2 459.0874} C_DIS
LIN {X 96.3414,Y -12.6793,Z 97,A -11.7383,B 24.9264,C -1.9807,E1 25.1586,E2 456.9859} C_DIS
LIN {X 96.7241,Y -9.3266,Z 97,A -9.6746,B 24.9257,C -1.9901,E1 25.1592,E2 454.9124} C_DIS
LIN {X 97.1046,Y -3.6546,Z 97,A -6.5681,B 24.9257,C -1.9912,E1 25.1597,E2 451.8218} C_DIS
LIN {X 97.1158,Y 3.3216,Z 97,A -2.0816,B 24.9236,C -2.0191,E1 25.1597,E2 447.2961} C_DIS
LIN {X 96.9263,Y 6.9149,Z 97,A -0.3571,B 24.9242,C -2.0102,E1 25.1593,E2 445.6028} C_DIS
LIN {X 96.6935,Y 9.643,Z 97,A 1.4366,B 24.9233,C -2.0224,E1 25.1588,E2 443.791} C_DIS
LIN {X 96.2839,Y 13.1187,Z 97,A 3.5283,B 24.9227,C -2.03,E1 25.1581,E2 441.6936} C_DIS
LIN {X 95.7421,Y 16.619,Z 97,A 5.6244,B 24.9222,C -2.0369,E1 25.1571,E2 439.5937} C_DIS
LIN {X 95.0668,Y 20.1258,Z 97,A 8.0888,B 24.9206,C -2.0576,E1 25.1557,E2 437.0947} C_DIS
LIN {X 94.3132,Y 23.4,Z 97,A 9.5983,B 24.9216,C -2.0451,E1 25.1547,E2 435.6235} C_DIS
LIN {X 93.4679,Y 26.5735,Z 97,A 11.9988,B 24.9197,C -2.0693,E1 25.1529,E2 433.1796} C_DIS
LIN {X 92.4536,Y 29.9118,Z 97,A 14.1519,B 24.9189,C -2.0792,E1 25.151,E2 431.0153} C_DIS
LIN {X 91.1703,Y 33.6227,Z 97,A 15.7754,B 24.9205,C -2.0589,E1 25.1495,E2 429.4489} C_DIS
LIN {X 90.4129,Y 35.6075,Z 97,A 17.3542,B 24.9192,C -2.0753,E1 25.1479,E2 427.8401} C_DIS
LIN {X 87.9536,Y 41.3119,Z 97,A 20.5312,B 24.9199,C -2.0667,E1 25.1444,E2 424.7006} C_DIS
LIN {X 86.8131,Y 43.66,Z 97,A 22.3263,B 24.9188,C -2.081,E1 25.1421,E2 422.8814} C_DIS
LIN {X 83.2807,Y 50.0693,Z 97,A 26.5409,B 24.9182,C -2.0887,E1 25.1363,E2 418.6706} C_DIS
LIN {X 80.1486,Y 54.9445,Z 97,A 30.0345,B 24.9173,C -2.1004,E1 25.131,E2 415.1667} C_DIS
LIN {X 78.1876,Y 57.6994,Z 97,A 32.0287,B 24.9169,C -2.1054,E1 25.1277,E2 413.1704} C_DIS
LIN {X 76.0451,Y 60.4949,Z 97,A 33.8842,B 24.9171,C -2.1019,E1 25.1245,E2 411.3319} C_DIS
LIN {X 73.7224,Y 63.3051,Z 97,A 35.9045,B 24.9171,C -2.1019,E1 25.1209,E2 409.3208} C_DIS
LIN {X 70.672,Y 66.6924,Z 97,A 38.7376,B 24.9162,C -2.1135,E1 25.1156,E2 406.4728} C_DIS
LIN {X 68.4014,Y 69.0193,Z 97,A 40.8379,B 24.9153,C -2.1246,E1 25.1114,E2 404.3552} C_DIS
LIN {X 65.6563,Y 71.6355,Z 97,A 43.7009,B 24.913,C -2.1532,E1 25.1054,E2 401.4363} C_DIS
LIN {X 62.3082,Y 74.5664,Z 97,A 45.2576,B 24.9159,C -2.1176,E1 25.1023,E2 399.9699} C_DIS
LIN {X 59.9758,Y 76.4553,Z 97,A 47.3962,B 24.9145,C -2.1348,E1 25.0975,E2 397.7986} C_DIS
LIN {X 56.6855,Y 78.9255,Z 97,A 49.458,B 24.9153,C -2.1253,E1 25.093,E2 395.7666} C_DIS
LIN {X 54.7483,Y 80.2815,Z 97,A 52.0692,B 24.9114,C -2.1736,E1 25.0867,E2 393.05} C_DIS
LIN {X 50.4594,Y 83.0436,Z 97,A 54.1629,B 24.9138,C -2.1436,E1 25.0819,E2 391.0338} C_DIS
LIN {X 44.5289,Y 86.3695,Z 97,A 57.96,B 24.914,C -2.1411,E1 25.0727,E2 387.2536} C_DIS
LIN {X 41.7037,Y 87.7688,Z 97,A 60.0632,B 24.9131,C -2.1525,E1 25.0673,E2 385.1291} C_DIS
LIN {X 36.7878,Y 89.9393,Z 97,A 63.4446,B 24.9122,C -2.1638,E1 25.0586,E2 381.7289} C_DIS
LIN {X 33.128,Y 91.3507,Z 97,A 65.514,B 24.9127,C -2.1569,E1 25.0532,E2 379.6801} C_DIS
LIN {X 29.3682,Y 92.6293,Z 97,A 68.0101,B 24.9121,C -2.1645,E1 25.0466,E2 377.1708} C_DIS
LIN {X 25.1876,Y 93.851,Z 97,A 70.2812,B 24.9129,C -2.1554,E1 25.0405,E2 374.925} C_DIS
LIN {X 21.9524,Y 94.6599,Z 97,A 72.8451,B 24.911,C -2.1783,E1 25.0334,E2 372.3105} C_DIS
LIN {X 18.4309,Y 95.408,Z 97,A 74.0208,B 24.9137,C -2.1449,E1 25.0305,E2 371.2155} C_DIS
LIN {X 15.8708,Y 95.8673,Z 97,A 75.983,B 24.9124,C -2.1608,E1 25.0249,E2 369.2175} C_DIS
LIN {X 12.3361,Y 96.3859,Z 97,A 78.0531,B 24.9124,C -2.16,E1 25.0192,E2 367.1511} C_DIS
LIN {X 8.8076,Y 96.7721,Z 97,A 80.1452,B 24.9124,C -2.1603,E1 25.0134,E2 365.0598} C_DIS
LIN {X 5.4098,Y 97.0213,Z 97,A 82.1681,B 24.9124,C -2.1608,E1 25.0078,E2 363.0365} C_DIS
LIN {X 1.3413,Y 97.1637,Z 97,A 85.3199,B 24.9103,C -2.1874,E1 24.9988,E2 359.822} C_DIS
LIN {X -2.9962,Y 97.1258,Z 97,A 87.1011,B 24.9126,C -2.159,E1 24.994,E2 358.1081} C_DIS
LIN {X -6.442,Y 96.9583,Z 97,A 89.4768,B 24.9117,C -2.1703,E1 24.9873,E2 355.7047} C_DIS
LIN {X -10.4979,Y 96.604,Z 97,A 91.6609,B 24.9124,C -2.1614,E1 24.9813,E2 353.5407} C_DIS
LIN {X -14.029,Y 96.1546,Z 97,A 93.7695,B 24.9124,C -2.1604,E1 24.9755,E2 351.4327} C_DIS
LIN {X -18.32,Y 95.4294,Z 97,A 95.8315,B 24.914,C -2.1409,E1 24.9699,E2 349.4149} C_DIS
LIN {X -20.1603,Y 95.0593,Z 97,A 97.4325,B 24.9127,C -2.1571,E1 24.9654,E2 347.7736} C_DIS
LIN {X -23.3461,Y 94.3263,Z 97,A 100.0344,B 24.9109,C -2.1789,E1 24.9582,E2 345.1163} C_DIS
LIN {X -27.5607,Y 93.1816,Z 97,A 101.8062,B 24.9135,C -2.1481,E1 24.9537,E2 343.4148} C_DIS
LIN {X -32.6295,Y 91.5311,Z 97,A 105.1063,B 24.9133,C -2.1497,E1 24.9449,E2 340.1047} C_DIS
LIN {X -36.2869,Y 90.1432,Z 97,A 107.0891,B 24.9145,C -2.1355,E1 24.9398,E2 338.1515} C_DIS
LIN {X -39.5224,Y 88.7725,Z 97,A 109.4678,B 24.9139,C -2.143,E1 24.9337,E2 335.7494} C_DIS
LIN {X -42.7929,Y 87.2429,Z 97,A 112.5543,B 24.9115,C -2.1725,E1 24.9258,E2 332.5844} C_DIS
LIN {X -47.4906,Y 84.7765,Z 97,A 115.7236,B 24.9118,C -2.1685,E1 24.918,E2 329.4156} C_DIS
LIN {X -52.1775,Y 81.9758,Z 97,A 117.6753,B 24.9158,C -2.1193,E1 24.9137,E2 327.575} C_DIS
LIN {X -54.7456,Y 80.2829,Z 97,A 120.0112,B 24.9146,C -2.1334,E1 24.9081,E2 325.1977} C_DIS
LIN {X -60.2287,Y 76.2555,Z 97,A 123.72,B 24.9161,C -2.1148,E1 24.8999,E2 321.5199} C_DIS
LIN {X -62.0269,Y 74.8002,Z 97,A 125.4668,B 24.9153,C -2.1246,E1 24.8961,E2 319.743} C_DIS
LIN {X -65.6479,Y 71.6432,Z 97,A 128.1467,B 24.9163,C -2.113,E1 24.8906,E2 317.0802} C_DIS
LIN {X -69.1719,Y 68.2469,Z 97,A 130.7477,B 24.9176,C -2.0966,E1 24.8854,E2 314.5072} C_DIS
LIN {X -71.9682,Y 65.2916,Z 97,A 133.4491,B 24.9172,C -2.1007,E1 24.8803,E2 311.7843} C_DIS
LIN {X -74.6479,Y 62.2101,Z 97,A 135.8261,B 24.9178,C -2.0934,E1 24.876,E2 309.4137} C_DIS
LIN {X -77.2294,Y 58.9761,Z 97,A 138.3106,B 24.9182,C -2.0884,E1 24.8717,E2 306.9294} C_DIS
LIN {X -80.8024,Y 53.9787,Z 97,A 141.6955,B 24.9196,C -2.0706,E1 24.8663,E2 303.5703} C_DIS
LIN {X -82.9845,Y 50.5566,Z 97,A 143.8416,B 24.9207,C -2.0558,E1 24.8632,E2 301.4487} C_DIS
LIN {X -84.3931,Y 48.1688,Z 97,A 146.1113,B 24.9195,C -2.0719,E1 24.8599,E2 299.1288} C_DIS
LIN {X -87.2653,Y 42.7478,Z 97,A 149.696,B 24.9204,C -2.0601,E1 24.8553,E2 295.5531} C_DIS
LIN {X -88.9599,Y 39.0974,Z 97,A 151.9365,B 24.9213,C -2.0486,E1 24.8528,E2 293.3276} C_DIS
LIN {X -91.2467,Y 33.4132,Z 97,A 155.6876,B 24.9218,C -2.0421,E1 24.849,E2 289.5712} C_DIS
Enddeposition()
END
